	15:	IF bAutoModeOn AND bIUnitA_RowStopperEnd  THEN
		bQAUnitA_RowStopperMotorFwd2:=FALSE;
		CTU_2.RESET:=TRUE;
		 step:=step+1;
		END_IF

	16:	step:=step+1;

	17:	tRowStopperRevDly1(IN:=TRUE , PT:=t#1.5s , Q=> , ET=> );
		IF tRowStopperRevDly1.Q THEN bQAUnitA_RowStopperMotorFwd1:=FALSE; step:=step+1; END_IF

	18:	 step:=step+1;


	19:	IF bAutoModeOn   THEN
		bAConvSecStart:=TRUE;
		bQAUnitA_RowStopperMotorRev1:=TRUE;
		CTU_2.RESET:=FALSE;
		step:=step+1;
		END_IF

	20:	IF bAutoModeOn  AND bIUnitB_LiftPistonHome THEN
		CountResetBit1_24:=TRUE;
		step:=step+1;
		END_IF

	21:	IF bAutoModeOn  AND bIUnitA_RowStopperHome THEN
		bQAUnitA_RowStopperMotorRev1:=FALSE;
		sRetreivalAStatus:= 'IDLE';
		step:=step+1;
		END_IF

	22:	IF bAutoModeOn (* AND( UnitACompleteCheckCount.CV =  iATotalNoOfCones)*) THEN
		(*bUnitARowStopperStarted:=FALSE;
		UnitACompleteCheckCount.RESET:=TRUE;*);
		bQAUnitA_RowStopperMotorRev1:=FALSE;
		step:=0;
		END_IF

END_CASE


				              		(* ################### 2*4 Sequence for  Count Check ##################*)



CASE step2 OF

	0:	IF bUnitARowStopperStarted   AND bAutoModeOn  THEN
		F_TRIG_3_24(CLK:=bIUnitBConeCrossing , Q=> );
		IF F_TRIG_3_24.Q THEN TON_6(IN:= FALSE); step2:=step2+1; END_IF END_IF


	1:	TON_6(IN:= FALSE); TON_9(IN:= FALSE); step2:=step2+1;

	2:	 bAUnitBConeCrossing_1_24 :=TRUE;  step2:=Step2+1;

	3: 	TON_6(IN:=  TRUE  , PT:=t#100ms,Q=> , ET=> );
		IF TON_6.Q THEN bAUnitBConeCrossing_1_24:=FALSE;   step2:=step2+1; END_IF

	4:	IF   bIUnitBConeCrossing   THEN
		TON_9(IN:=  TRUE  , PT:=t#50ms,Q=> , ET=>);
		IF TON_9.Q THEN TON_6(IN:= FALSE);  step2:=step2+1; END_IF END_IF

	5:	TON_9(IN:= FALSE);
		step2:=0;

END_CASE


CASE step4 OF

	0:	IF bUnitARowStopperStarted    AND bAutoModeOn THEN
		F_TRIG_5(CLK:=bIUnitAConeCrossing , Q=> );
		IF F_TRIG_5.Q THEN TON_8(IN:= FALSE); step4:=step4+1; END_IF END_IF


	1:	TON_8(IN:= FALSE);
		TON_10(IN:= FALSE);
		step4:=step4+1;


	2:	 bAUnitAConeCrossing_1_24 :=TRUE;
		 step4:=step4+1;

	3: 	TON_8(IN:=  TRUE  , PT:=t#100ms,Q=> , ET=> );
		IF TON_8.Q   THEN  bAUnitAConeCrossing_1_24:=FALSE;  step4:=step4+1; END_IF

	4:	IF   bIUnitAConeCrossing   THEN
		TON_10(IN:=  TRUE  , PT:=t#50ms,Q=> , ET=>);
		IF TON_10.Q THEN TON_8(IN:= FALSE);  step4:=step4+1; END_IF END_IF

	5:	TON_8(IN:= FALSE);
		step4:=0;

END_CASE



UnitAConeCrossCount(
	CU:= bAUnitAConeCrossing_1_24   ,
	RESET:= ,
	PV:=3 ,
	Q=> ,
	CV=> );


UnitACompleteCheckCount(
	CU:=  bAUnitBConeCrossing_1_24   ,
	RESET:= ,
	PV:=iATotalNoOfCones ,
	Q=> ,
	CV=>UnitACompleteCheckCountCV );



						(*============= After 24 Cone Crossed the UnitB limit switch==============*)


IF UnitACompleteCheckCount.CV >=  iATotalNoOfCones AND CountResetBit1_24    THEN
 tConeCrossDly(IN:=TRUE , PT:=t#0.3s , Q=> , ET=> );  END_IF

IF tConeCrossDly.Q   THEN
tConeCrossDly_1_24(IN:=TRUE , PT:=t#1s , Q=> , ET=> );
UnitACompleteCheckCount.RESET:=TRUE;
bQAUnitA_RowStopperMotorFwd2:=FALSE;
bQAUnitA_RowStopperMotorFwd1:=FALSE;

IF tConeCrossDly_1_24.Q THEN
 bUnitARowStopperStarted:=FALSE;
UnitACompleteCheckCount.RESET:=TRUE;
 tConeCrossDly(IN:=FALSE);
tConeCrossDly_1_24(in:=FALSE);
CountResetBit1_24:=FALSE;
bQAUnitA_RowStopperMotorFwd2:=FALSE;
bQAUnitA_RowStopperMotorFwd1:=FALSE;
(*step:=0;*)
END_IF
IF tConeCrossDly_1_24.Q AND bIUnitA_RowStopperHome THEN
		bQAUnitA_RowStopperMotorRev1:=FALSE;
END_IF

END_IF


IF b2_3SetHmiSelected THEN iATotalNoOfCones:=18; END_IF
IF b2_4SetHmiSelected THEN iATotalNoOfCones:=24; END_IF

(*===============Stop Sequence===========*)


IF NOT bIEmergencySwitch OR bIMcStop OR bServoOff OR   bStopHmi THEN bStopRetUnitA:=TRUE;  UnitACompleteCheckCount.RESET:=TRUE;END_IF


IF bStopRetUnitA THEN
step:=0;
bAUnitAWeighOk:=FALSE;
bAConvFirstStart:=FALSE;
bQAUnitA_RowStopperMotorFwd1:=FALSE;
UnitAConeCrossCount.RESET:=FALSE;
bQAUnitA_RowStopperMotorFwd2:=FALSE;
bAConvSecStart:=FALSE;
bQAUnitA_RowStopperMotorRev1:=FALSE;
bRetUnitARst:=TRUE;
bUnitARowStopperStarted:=FALSE;
		UnitACompleteCheckCount.RESET:=FALSE;
step4:=0;
step2:=0;
END_IF

IF bIUnitA_RowStopperHome THEN
bStopRetUnitA:=FALSE;
bRetUnitARst:=FALSE;
END_IF

IF bRetUnitARst THEN
step4:=0;
step2:=0;
 END_IF


(***HMI Count***)

IF bUnitARowStopperStarted THEN
 RowStopperCountvalue:=UnitACompleteCheckCountCV;

ELSIF  NOT bUnitARowStopperStarted THEN
RowStopperCountvalue:=0;

END_IF
Count_Hmi:=RowStopperCountvalue;
END_PROGRAM

(* POU FunctionBlocks/SenSelect, ST *)
FUNCTION_BLOCK SenSelect
VAR_INPUT


	bVarIn1: BOOL;
	bVarIn2: BOOL;
	bVarIn3: BOOL;
	bVarIn4: BOOL;
END_VAR
VAR_OUTPUT


	ByteResult: USINT;
END_VAR
VAR

END_VAR
ByteResult.0:=bVarIn1;
ByteResult.1:=bVarIn2;
ByteResult.2:=bVarIn3;

ByteResult;
END_FUNCTION_BLOCK

(* POU Auto1/UnitB_RowStopper24, ST *)
PROGRAM UnitB_RowStopper24
VAR




	step: INT;
	bAUnitAWeighOk: BOOL;
	CTU_1: CTU;
	CTU_1Enable: BOOL;
	R_TRIG_1: R_TRIG;
	R_TRIG_2: F_TRIG;
	bQAUnitA_RowStopperMotorFwd1: BOOL;
	bQAUnitA_RowStopperMotorFwd2: BOOL;
	tRowStopperRevDly1: TON;
	bQAUnitA_RowStopperMotorRev1: BOOL;
	CTU_2: CTU;
	UnitBConeCount: CTU;
	CTU_1EnableUnitB: BOOL;
	temp1: BOOL;
	bStopRetUnitB: BOOL;
	bRetUnitBRst: BOOL;
	RowStopperMotorStopDly: TON;
	F_TRIG_3: F_TRIG;

	UnitBOverTemp: BOOL;
	bStartTemp1: BOOL;
	R_TRIG_5: R_TRIG;
	test: BOOL;
	bStopTemp2: BOOL;
	CTU_2CV: INT;
	CTU_test: CTU;
	R_TRIG_test: R_TRIG;
	InterLockStep: INT;

	CTU_2Enable: BOOL;
	timer1: TON;
	UnitBCompleteCheckCountCV: INT;
	Ctu_2_Rst: BOOL;
	F_TRIG_1: F_TRIG;
	bRestBit: BOOL;
	bResetBit: BOOL;
	R_TRIG_6: R_TRIG;
	timer2: TON;
	SenSelect_2: SenSelect;
	iSensorOnVal: UINT;
	iAConeCrossCount1: INT;
	GetDLy: TON;
	bCheckSensor1: BOOL;
	step2: INT;
	TON_9: TON;
	TON_6: TON;
	tConeCrossDly: TON;
	bAUnitBConeCrossing_24_B: BOOL;
	tConeCrossDly_2_24: TON;
	CountResetBit2_24: BOOL;
END_VAR
(*=============Checking the No of sensors sensed================*)

IF bCheckSensor1 THEN
SenSelect_2(
		bVarIn1:=bIUnitBConedetection1 ,
		bVarIn2:= bIUnitBConedetection2,
		bVarIn3:= bIUnitBConedetection3,
		ByteResult=>iSensorOnVal );
END_IF

IF iSensorOnVal=7 THEN iAConeCrossCount1:=3;
	ELSIF  iSensorOnVal=6 THEN iAConeCrossCount1:=2;
	ELSIF  iSensorOnVal=5 THEN iAConeCrossCount1:=2;
	ELSIF  iSensorOnVal=4 THEN iAConeCrossCount1:=1;
	ELSIF  iSensorOnVal=3 THEN iAConeCrossCount1:=2;
	ELSIF  iSensorOnVal=2 THEN iAConeCrossCount1:=1;
	ELSIF  iSensorOnVal=1 THEN iAConeCrossCount1:=1;
END_IF


bQAUnitB_RowStopperMotorForward:=( bQAUnitB_RowStopperMotorFwd1 OR bQAUnitB_RowStopperMotorFwd2  );

bQAUnitB_RowStopperMotorReverse:= ( bQAUnitB_RowStopperMotorRev1 OR bRetUnitBRst  );


CASE step OF

	0:	IF bAutoModeOn AND bAUnitBWeighOk  AND bRetUnitBStart  AND NOT bStopEnable AND bAinterlockinit   THEN
		UnitBConeCrossCount.RESET:=TRUE;
		CTU_2.RESET:=TRUE;
		UnitBCompleteCheckCount_24.RESET:=TRUE;
		CountResetBit2_24 :=FALSE;
		step:=step+1;
		END_IF

	1:	 step:=step+1;

	2:	IF bAutoModeOn   AND  UnitBCompleteCheckCount_24.CV = 0 AND NOT CountResetBit2_24 THEN
		CTU_2.RESET:=FALSE;
		UnitBConeCrossCount.RESET:=FALSE;
		UnitBCompleteCheckCount_24.RESET:=FALSE;
		step:=step+1;
		END_IF


	3:	bRestBit:=TRUE;
		step:=step+1;


	4:	IF bAutoModeOn  AND NOT bIUnitBConedetection1 AND NOT bIUnitBConedetection2 AND NOT bIUnitBConedetection3
		AND NOT bUnitARowStopperStarted AND NOT bAMainIntStarted  AND NOT bStopEnable AND NOT bAPauseSeq THEN
		timer1(IN:=FALSE);
		timer2(IN:=FALSE);
		bAConvFirstStartUnitB:=TRUE;
		bQAUnitB_RowStopperMotorFwd1:=TRUE;
		bAUnitBWeighOk:=FALSE;
		bRetUnitBStart:=FALSE;
		sRetreivalBStatus:= 'Running';
		bUnitBRowStopperStarted:=TRUE;
		step:=step+1;
		ELSIF   bIUnitB_RowStopperEnd  THEN  step:=12;
		END_IF

	5:	RowStopperMotorStopDly(In:=FALSE); step:=step+1;


	6:	IF bIUnitBConedetection1 OR  bIUnitBConedetection2  OR  bIUnitBConedetection3 THEN
		UnitBConeCount.RESET:=TRUE;
		step:=step+1;
		ELSIF NOT bIUnitBConedetection1 AND NOT  bIUnitBConedetection2 AND NOT  bIUnitBConedetection3 AND bIUnitB_RowStopperEnd THEN
		step:=15;
		END_IF

	7:	RowStopperMotorStopDly( IN:=TRUE , PT:=T#0.5S , Q=> , ET=> );IF RowStopperMotorStopDly.Q   THEN  step:=step+1; END_IF


	8:	UnitBConeCount.RESET:=FALSE;
		bQAUnitB_RowStopperMotorFwd1:=FALSE;
		tRowStopperRevDly1(IN:=FALSE);
		step:=step+1;

	9:	IF NOT bAPauseSeq THEN bCheckSensor1:=TRUE;  step:=step+1; END_IF

	10:	GetDLy(IN:=TRUE , PT:=t#0.6s , Q=> , ET=> );
		 IF GetDLy.Q THEN bCheckSensor1:=FALSE;   step:=step+1;
		END_IF


	11:	IF  (UnitBConeCount.CV=iAConeCrossCount1)  AND NOT bIUnitB_RowStopperEnd THEN
		RowStopperMotorStopDly(In:=FALSE);
		 step:=4;
		ELSE
		IF bIUnitB_RowStopperEnd THEN
		    step:=step+1;
		END_IF END_IF



	12:	IF NOT bAPauseSeq THEN tRowStopperRevDly1(IN:=FALSE); step:=step+1; END_IF

	13:	IF bAutoModeOn    (* AND NOT bQAFeedingConveyorMotor *) THEN
		bQAUnitB_RowStopperMotorFwd2:=TRUE;
		step:=step+1;
		END_IF


	14:	 step:=step+1;

	15:	IF bAutoModeOn AND bIUnitB_RowStopperEnd THEN
		bQAUnitB_RowStopperMotorFwd2:=FALSE;
		bQAUnitB_RowStopperMotorFwd1:=FALSE;
		UnitBConeCount.RESET:=TRUE;
		CTU_2.RESET:=TRUE;
		 step:=step+1;
		END_IF

	16:	  step:=step+1;

	17:	tRowStopperRevDly1(IN:=TRUE , PT:=t#1.5s , Q=> , ET=> );
		IF tRowStopperRevDly1.Q THEN step:=step+1; END_IF

	18:	step:=step+1;

	19:	IF bAutoModeOn  THEN
		bAConvSecStartUnitB:=TRUE;
		CTU_2.RESET:=FALSE;
		UnitBConeCount.RESET:=FALSE;
		bQAUnitB_RowStopperMotorRev1:=TRUE;
		step:=step+1;
		END_IF

	20:	IF bAutoModeOn  AND bIUnitB_LiftPistonEnd THEN
		CountResetBit2_24:=TRUE;
		step:=step+1;
		END_IF


	21:	IF bAutoModeOn  AND bIUnitB_RowStopperHome THEN
		bQAUnitB_RowStopperMotorRev1:=FALSE;
		sRetreivalBStatus:= 'IDLE';
		step:=step+1;
		END_IF

	22:	IF bAutoModeOn  (*AND (UnitBCompleteCheckCount_24.CV >=  iATotalNoOfCones)*) THEN
 		(*bUnitBRowStopperStarted:=FALSE;
		UnitBCompleteCheckCount_24.RESET:=FALSE;*)
		step:=0;
		END_IF



END_CASE


					(* ######################### 2*4 Cone Count Sequence ####################*)




CASE step2 OF

	0:	IF bUnitBRowStopperStarted  AND bAutoModeOn THEN
		F_TRIG_3(CLK:=bIUnitBConeCrossing , Q=> );
		IF F_TRIG_3.Q THEN TON_6(IN:= FALSE); step2:=step2+1; END_IF END_IF


	1:	TON_6(IN:= FALSE);
		TON_9(IN:= FALSE);
		step2:=step2+1;


	2:	 bAUnitBConeCrossing_24_B :=TRUE;
		 step2:=Step2+1;

	3:	 step2:=step2+1;

	4: 	TON_6(IN:=  TRUE  , PT:=t#100ms,Q=> , ET=> );
		IF TON_6.Q THEN bAUnitBConeCrossing_24_B:=FALSE;   step2:=step2+1; END_IF


	5:	 step2:=step2+1;

	6:	IF   bIUnitBConeCrossing THEN
		TON_9(IN:=  TRUE  , PT:=t#50ms,Q=> , ET=>);
		IF TON_9.Q THEN TON_6(IN:= FALSE);  step2:=step2+1; END_IF END_IF


	7:	 step2:=step2+1;

	8:	 step2:=step2+1;

	9:	 step2:=step2+1;

	10:	TON_9(IN:= FALSE);
		step2:=0;


END_CASE




UnitBConeCount(
	CU:= ( bAUnitBConeCrossing_24_B)  ,
	RESET:= ,
	PV:=3 ,
	Q=> ,
	CV=> );

UnitBCompleteCheckCount_24(
	CU:= bAUnitBConeCrossing_24_B  ,
	RESET:= ,
	PV:=iATotalNoOfCones ,
	Q=> ,
	CV=>UnitBCompleteCheckCountCV );

(*============= After 18 Cone Crossed the UnitB limit switch==============*)

IF UnitBCompleteCheckCount_24.CV >=  iATotalNoOfCones AND CountResetBit2_24  AND bAutoModeOn  THEN
 tConeCrossDly(IN:=TRUE , PT:=t#0.3s , Q=> , ET=> );
END_IF

IF tConeCrossDly.Q THEN
tConeCrossDly_2_24(IN:=TRUE , PT:=t#1s , Q=> , ET=> );
UnitBCompleteCheckCount_24.RESET:=TRUE;

IF tConeCrossDly_2_24.Q THEN
 bUnitBRowStopperStarted:=FALSE;
UnitBCompleteCheckCount_24.RESET:=TRUE;
  tConeCrossDly(IN:=FALSE);
tConeCrossDly_2_24(in:=FALSE);
CountResetBit2_24:=FALSE;
 END_IF
ELSE
UnitBCompleteCheckCount.RESET:=FALSE;

END_IF







(*===============Stop Sequence===========*)


IF NOT bIEmergencySwitch OR bIMcStop OR bServoOff OR  bStopHmi THEN bStopRetUnitB:=TRUE; END_IF


IF bStopRetUnitB THEN
step:=0;
bAUnitBWeighOk:=FALSE;
bAConvFirstStartUnitB:=FALSE;
bQAUnitB_RowStopperMotorFwd1:=FALSE;
UnitBConeCount.RESET:=FALSE;
bQAUnitB_RowStopperMotorFwd2:=FALSE;
bAConvSecStartUnitB:=FALSE;
bQAUnitB_RowStopperMotorRev1:=FALSE;
bRetUnitBRst:=TRUE;
bUnitBRowStopperStarted:=FALSE;
step2:=0;
END_IF

IF bIUnitB_RowStopperHome THEN
bStopRetUnitB:=FALSE;
bRetUnitBRst:=FALSE;
END_IF



IF bAutoModeOn  AND  bResetBit AND bIUnitBConedetection1 AND bIUnitBConedetection3 AND bIUnitBConedetection3
AND NOT  bIUnitB_RowStopperHome THEN Ctu_2_Rst:=TRUE;  ELSE Ctu_2_Rst:= FALSE; END_IF

R_TRIG_6(CLK:=Ctu_2_Rst , Q=> );

CTU_2.RESET:= R_TRIG_6.Q;


(***HMI Count***)

IF bUnitBRowStopperStarted THEN
CountB_Hmi:=UnitBCompleteCheckCountCV;
ELSIF  NOT bUnitBRowStopperStarted THEN
CountB_Hmi:=0;
END_IF
END_PROGRAM

(* POU Auto/OneMinConv, ST *)
	PROGRAM OneMinConv
VAR
	bQAGrossWtPiston1: BOOL;
	bQARollerConvMotor1: BOOL;
	step: INT;
	Timer1: TON;
	Timer2: TON;

	Timer3: TON;
	bQARollerConvMotor2: BOOL;
	bAPartCount: BOOL;
	R_TRIG_1: R_TRIG;
	PartCounter: CTU;
	rGrossWtTolMax: REAL;
	rGrossWtTolMin: REAL;
	bGrossWieghtOkTemp: BOOL;
	rGrossWeighToReportTemp: STRING;
	iTotalpartCounttemp: DINT;
END_VAR
	bQAGrossWtPiston:= bQAGrossWtPiston1 ;
	bQARollerConvMotor:=bQARollerConvMotor1 OR bQARollerConvMotor2 ;


rGrossWtTolMax:= (sSettingArray[i].iGrosswt + sSettingArray[i].iGrossTol);

rGrossWtTolMin:= (sSettingArray[i].iGrosswt - sSettingArray[i].iGrossTol);


CASE step OF

	0:	IF bAutoModeOn AND bAOneMinConvStart   AND NOT bAPauseSeq THEN
		bQARollerConvMotor1:=TRUE;
		Timer1(IN:=FALSE);
		Timer2(IN:=FALSE);
		Timer3(IN:=FALSE);
		 step:=step+1;
		END_IF

	1:	IF bIGrossWtDeductSensor THEN
		bQARollerConvMotor1:=FALSE;
		bAOneMinConvStart:=FALSE;
		 step:=step+1;
		END_IF

	2:	Timer1(IN:=TRUE , PT:=t#1s , Q=> , ET=> );
		IF Timer1.Q THEN step:= step+1; END_IF   (*====== Modified for  Gross  Weight   bypass  then removed  ==============*)

	3:	bQAGrossWtPiston1:=TRUE;
		IF bIGrossWtPistonEnd  AND NOT bAGrossWtSenRsError THEN step:=step+1; END_IF

	4:	 tGrossWtCheckDly(IN:=FALSE);
		Timer2(IN:=TRUE , PT:=t#1s , Q=> , ET=> );
		IF Timer2.Q THEN step:=step+1; END_IF

	5:	bReadGWieght:=TRUE;
		step:=step+1;


	6:	IF bReadGWieght THEN
		tGrossWtCheckDly(IN:=TRUE , PT:=t#9.5s , Q=> , ET=> );
		IF tGrossWtCheckDly.Q THEN 	step:=step+1;END_IF
		END_IF


	7:	IF  rGrossWeight >=rGrossWtTolMin  AND   rGrossWeight  <= rGrossWtTolMax  THEN
		bGrossWieghtOkTemp:=TRUE; rGrossWeighToReport:=rGrossWeight ;  bGrossWieghtNokTemp:=FALSE;
		step:=step+1;
		ELSIF  rGrossWeight  >= rGrossWtTolMax THEN
		bGrossWieghtNokTemp:=TRUE; bGrossWieghtOkTemp:=FALSE;
		step:=step+2;
		ELSIF   rGrossWeight  <=rGrossWtTolMin   THEN
		bGrossWieghtNokTemp:=TRUE; bGrossWieghtOkTemp:=FALSE;
		step:=step+2;
		END_IF


	8:	IF bGrossWieghtOkTemp THEN bGrossWieghtOk:=TRUE; bQAGrossWieghtOkIndi:=TRUE; step:=step+2;  END_IF

	9:	IF bGrossWieghtNokTemp THEN bGrossWieghtNOk:=TRUE; bReadGWieght:=FALSE; step:=step+2; END_IF


	10:	IF bGrossWieghtOk (*  AND NOT bGrossWieghtNok *) AND bAutoModeOn  AND NOT bAPauseSeq THEN bQAGrossWtPiston1:=FALSE; bReadGWieght:=FALSE; bGrossWieghtOkTemp:=FALSE; bQAGrossWieghtOkIndi:=FALSE;   (*====== Modified for  Gross  Weight   bypass  ==============*)
		bACyclePass:=TRUE;
		GrossWtReedSwBit:=TRUE;
		step:=step+2;
		 END_IF

	11:	IF bErrorReset THEN  bGrossWieghtNOk:=FALSE;  step:=4; END_IF

	12:	IF bIGrossWtPistonHome  AND NOT bAGrossWtHomeSenRsError THEN GrossWtReedSwBit:=FALSE ;step:=step+1;END_IF

	13:	bACyclePass:=FALSE;
		 step:=step+1;

	14:	IF NOT   bAPauseSeq  THEN
		bQARollerConvMotor2:=TRUE;
		bReadGWieght:=FALSE;
		Step:=Step+1;
	(*	Timer3(IN:=TRUE , PT:=t#30s , Q=> , ET=> );
		IF Timer3.Q THEN step:=step+1; END_IF    *)
		END_IF


	15:	IF NOT  bIGrossWtDeductSensor THEN
		bQARollerConvMotor2:=FALSE;
		 bOneMinConvOver:=TRUE;

		step:=0;
		END_IF

END_CASE

sFinalGrossWt:=MID(STR:=rGrossWeighToReportTemp, LEN:=7, POS:=1);

rGrossWeighToReportTemp:=REAL_TO_STRING (rGrossWeight);

IF bGrossWieghtOk THEN var_7:= sFinalGrossWt ; END_IF

(*=====Carton Completed Count Logic=========*)

	IF bACyclePass AND bAutoModeOn THEN bAPartCount:=TRUE; ELSE bAPartCount:=FALSE; END_IF


R_TRIG_1(CLK:=bAPartCount , Q=> );
PartCounter(
	CU:=R_TRIG_1.Q ,
	RESET:=bSaveRecipeHmi ,
	PV:= 9999,
	Q=> ,
	CV=> );

iTotalpartCountTemp:=PartCounter.CV;

ITotalSample:=iTotalpartCountTemp;
(*========== No Of Cartons Processed Logic==========*)

IF b2_3SetHmiSelected AND bACyclePass THEN   iTotalCones := ( iTotalpartCountTemp  * 18 );  iTotalpartCount:=iTotalpartCountTemp;

ELSIF b2_4SetHmiSelected  AND bACyclePass THEN  iTotalCones := ( iTotalpartCountTemp  * 24  );  iTotalpartCount:=iTotalpartCountTemp;

END_IF


IF NOT bIEmergencySwitch OR   bStopHmi   OR bServoOff  OR bIMcStop  THEN
step:=0;
bReadGWieght:=FALSE;
bAOneMinConvStart:=FALSE;
bQARollerConvMotor1:=FALSE;
bQARollerConvMotor2:=FALSE;
bQAGrossWtPiston1:=FALSE;
bGrossWieghtNOk:=FALSE;
bACyclePass:=FALSE;
Timer1(IN:=FALSE);
Timer2(IN:=FALSE);
Timer3(IN:=FALSE);
tGrossWtCheckDly(IN:=FALSE);
END_IF
END_PROGRAM

(* POU Auto/Sealing_Unit, ST *)
PROGRAM Sealing_Unit
VAR
	step: INT;
	tA3ConeStartDly: TON;
	tA3ConeSealCompDly: TON;
	test: BOOL;

END_VAR
IF NOT bIEmergencySwitch OR  bStopHmi    OR bServoOff OR bIMcStop   THEN
	tA3ConeStartDly(IN:=FALSE);
	tA3ConeSealCompDly(IN:=FALSE);
	bQASealingSeparatorYAxisPistonValve:=FALSE;
	bQASealingTopPistonValve:=FALSE;
	bQASealingSeparatorXAxisPistonValve:=FALSE;
	bA3ConeWrappOver:=FALSE;
	bA3ConeWrappOver_24:=FALSE;
	bA4thWrappOver:=FALSE;
	bA6thConeWrappOver:=FALSE;
	bA8thConeWrappOver:=FALSE;
	bA6ConeWrappOver23:=FALSE;
	bMManualSealOn:=FALSE;
	bQMSealingTopPistonValve:=FALSE;
	Step:=0;
	SealingOver1:=FALSE;
	bA3ConeWrappOver_24:=FALSE;
END_IF


CASE step OF

	0:	IF b2_4SetHmiSelected OR b2_3SetHmiSelected  AND bAutoModeOn  THEN
		Step:=step+1;
		END_IF

	1:	step:=step+1;


	2:	IF bAutoModeOn AND  bA3ConeWrappOver  OR bA4thWrappOver OR bA6thConeWrappOver  OR bA8thConeWrappOver  OR bA6ConeWrappOver23
		OR bA3ConeWrappOver_24 AND NOT bAPauseSeq THEN
		tA3ConeStartDly(IN:=TRUE , PT:=t#1s , Q=> , ET=> );
		IF tA3ConeStartDly.Q THEN  step:=step+1; END_IF
		END_IF

	3:	IF bIWrappingChannelPiston1_Home AND bIWrappingChannelPiston2_Home  AND bIWrappingChannelPiston3_Home THEN
		step:=step+1;END_IF    sMessage_Sealing:='Check Wrapping Piston Home 1 & 2 & 3 Reed Switch';


	4:	IF bAutoModeOn AND   bISealingBottomPistonHome  AND bISealingTopPistonHome AND bISealingSeparatorXAxisHome
		AND bISealingSeparatorYAxisHome   AND  NOT bAPauseSeq THEN
		bQASealingSeparatorYAxisPistonValve:=TRUE;
		tA3ConeSealCompDly(IN:=FALSE);
		 step:=step+1;
		END_IF  sMessage_Sealing:='Check All  Piston Home  Reed Switch';

	5:	 step:=step+1;

	6:	IF bAutoModeOn AND  bISealingSeparatorYAxisEnd AND  NOT bAPauseSeq  AND NOT bASealSepaY_axisRsError  THEN
		tA3ConeStartDly(IN:=FALSE);
		bQASealingTopPistonValve:=TRUE;
		step:=step+1;
		END_IF

	7:	step:=step+1;

	8:	IF bAutoModeOn AND  bISealingTopPistonEnd AND bISealingBottomPistonEnd  THEN
		tA3ConeSealCompDly(IN:=TRUE, PT:= SealComDlyTemp, Q=> , ET=> );
		IF tA3ConeSealCompDly.Q THEN   step:=step+1; END_IF
		END_IF

	9:	step:=step+1;

	10:	IF bAutoModeOn AND  bISealingTopPistonEnd AND bISealingBottomPistonEnd AND bISealingSeparatorYAxisEnd AND  NOT bAPauseSeq
		  AND NOT SealTopBottomRsError THEN
		bQASealingSeparatorXAxisPistonValve:=TRUE;
		step:=step+1;
		END_IF  sMessage_Sealing:='Check Sealing Top, Bottom, Separator YAxis  Piston End  Reed Switch';

	11:	 step:=step+1;

	12:	IF bAutoModeOn AND  bISealingSeparatorXAxisEnd AND  NOT bAPauseSeq  AND  NOT bASealSepaX_axisRsError THEN
		step:=step+1;
		 END_IF

	13:	 step:=step+1;

	14:	bQASealingTopPistonValve:=FALSE;
		bA3ConeWrappOver:=FALSE;
		bA3ConeWrappOver_24:=FALSE;
		bA4thWrappOver:=FALSE;
		bA6thConeWrappOver:=FALSE;
		bA8thConeWrappOver:=FALSE;
		bA6ConeWrappOver23:=FALSE;
		bQASealingSeparatorYAxisPistonValve:=FALSE;
		bQASealingSeparatorXAxisPistonValve:=FALSE;
		step:=step+1;

	15:	step:=step+1;

	16:	IF b2_4SetHmiSelected THEN step:=step+1; ELSIF b2_3SetHmiSelected THEN step:=step+1; END_IF


	17:	IF bAutoModeOn AND NOT bA3ConeWrappOver AND NOT bA4thWrappOver AND NOT bA6thConeWrappOver AND NOT bA8thConeWrappOver
		AND NOT bA3ConeWrappOver_24 AND bISealingSeparatorXAxisHome AND  bISealingTopPistonHome AND bISealingBottomPistonHome
		AND bISealingSeparatorYAxisHome  THEN
		SealingOver1:=TRUE; step:=step+1;
		END_IF sMessage_Sealing:='Check All Piston Home  Reed Switch';


	18:	IF bAutoModeOn AND bISealingSeparatorXAxisHome AND  bISealingTopPistonHome AND bISealingBottomPistonHome AND bISealingSeparatorYAxisHome
		THEN
		 step:=step+1;
		END_IF sMessage_Sealing:='Check All Piston Home  Reed Switch';

	19:	step:=step+1;

	20:	 step:=step+1;

	21:	step:=0;



END_CASE



IF bAutoModeOn AND NOT bA3ConeWrappOver AND NOT bA4thWrappOver AND NOT bA6thConeWrappOver AND NOT bA8thConeWrappOver AND
 bISealingSeparatorXAxisHome AND  bISealingTopPistonHome AND bISealingBottomPistonHome AND bISealingSeparatorYAxisHome  THEN
SealingSafety:=TRUE; ELSE SealingSafety:=FALSE;END_IF
END_PROGRAM

(* POU New Folder/ConeAllignAlarm, ST *)
PROGRAM ConeAllignAlarm
VAR
	ConeMiss: INT;
	TON_1: TON;
	TON_2: TON;
	TON_3: TON;
	Timer_4: TON;

	bAConeMissErrorAtWrpConvTemp: BOOL;
	bNotSensing: BOOL;
	bNotSensingtEMP: BOOL;

	TON_3_24: TON;
	TON_12: TON;

END_VAR
(*...................Cone Allignment Alarm.....................*)


IF bQAWrappingConveyorMotor1 AND b2_3SetHmiSelected THEN TON_3(IN:=TRUE , PT:= t#7s, Q=> , ET=> );  ELSE  TON_3(IN:=FALSE); END_IF

IF  bAutoModeOn AND TON_3.Q AND NOT bIWrappingCone1 AND b2_3SetHmiSelected  THEN
 bAConeMissErrorAtWrpConvTemp:=TRUE;  END_IF

IF bAutoModeOn  AND bIWrappingCone1 AND b2_3SetHmiSelected THEN
bAConeMissErrorAtWrpConvTemp:=FALSE; END_IF     (*Change*)

IF bErrorReset AND b2_3SetHmiSelected THEN
TON_3(IN:=FALSE); bAConeMissErrorAtWrpConvTemp:=FALSE;  END_IF

IF NOT bIEmergencySwitch OR bStopHmi  OR bServoOff OR bIMcStop  AND b2_3SetHmiSelected  THEN
bAConeMissErrorAtWrpConvTemp:=FALSE;
ConeMissAlarm:='';
 TON_3(IN:=FALSE);
END_IF


(* ================== Cone Missing 2 & 3 Logic on Wrapping Conveyor===============*)

IF bWrapConvStopped2 AND b2_3SetHmiSelected  AND  NOT bAPauseSeq  THEN Timer_4(IN:=TRUE , PT:=t#4s , Q=> , ET=> ); ELSE  Timer_4(IN:=FALSE); END_IF

IF bAutoModeOn  AND  Timer_4.Q AND  (NOT bIWrappingCone1 OR NOT bIWrappingCone2 OR NOT bIWrappingCone3 ) AND NOT bConeMiss2AtWrapConvtEMP
AND b2_3SetHmiSelected  THEN bConeMiss2AtWrapConvtEMP:=TRUE;
ELSE
 IF  bAutoModeOn AND b2_3SetHmiSelected AND bWrapConvStopped2   AND bIWrappingCone1 AND bIWrappingCone2 AND bIWrappingCone3 THEN
  TON_12(IN:=TRUE , PT:= t#0.7s, Q=> , ET=> );  Timer_4(IN:=FALSE);

IF TON_12.Q AND b2_3SetHmiSelected THEN  bWrapConvStopped2:=FALSE; END_IF
 END_IF  END_IF


IF bErrorReset  AND bConeMiss2AtWrapConvtEMP AND  bIWrappingCone1 AND bIWrappingCone2 AND bIWrappingCone3
 THEN Timer_4(IN:=FALSE); TON_12(in:=FALSE); bConeMiss2AtWrapConvtEMP:=FALSE;
bAByPassOn:=TRUE;  bConeMiss2AtWrapConv:=FALSE; bConeMiss2AtWrapConvtEMP:=FALSE; ConeMissAlarm:=''; END_IF


IF NOT bIEmergencySwitch OR bIMcStop OR bStopHmi OR bServoOff THEN
bWrapConvStopped2:=FALSE;
bConeMiss2AtWrapConvtEMP:=FALSE;
bCount_ConvLockBit:=FALSE;
Timer_4(IN:=FALSE);
END_IF



(*============Wrapping Cone Missing Msg to Hmi=============*)

IF bAConeMissErrorAtWrpConvTemp AND b2_3SetHmiSelected THEN
ConeMissAlarm:='Allign the Cone  on Wrapping Conveyer ';
ELSIF bConeMiss2AtWrapConvtEMP AND b2_3SetHmiSelected  THEN
ConeMissAlarm:='Allign the Cone  on Wrapping Conveyer ';
ELSIF bConeMiss3AtWrapConv  AND b2_3SetHmiSelected THEN
ConeMissAlarm:='Allign the Cone  on Wrapping Conveyer ';
ELSIF bConeMiss4AtWrapConv AND b2_3SetHmiSelected  THEN
ConeMissAlarm:='Allign the Cone  on Wrapping Conveyer ';

ELSIF bACheckWrappConvError1_23 AND b2_3SetHmiSelected  THEN
ConeMissAlarm:='Check Wrapping Sensor 1 & 2 & 3';
ELSIF bACheckWrappConvError2  AND b2_3SetHmiSelected THEN
ConeMissAlarm:='Check Wrapping Sensor  2 & 3';
ELSIF bACheckWrappConvError3 AND b2_3SetHmiSelected THEN
ConeMissAlarm:='Check Wrapping Sensor 1 & 2 & 3';
ELSIF bACheckWrappConvError4 AND b2_3SetHmiSelected THEN
ConeMissAlarm:='Check Wrapping Sensor  3';
ELSIF NOT bConeMiss1AtWrapConv  AND NOT bAConeMissErrorAtWrpConvTemp AND NOT  bConeMiss2AtWrapConvtEMP AND NOT bConeMiss3AtWrapConv
AND NOT bConeMiss4AtWrapConv AND NOT  bACheckWrappConvError1_23 AND NOT bACheckWrappConvError2 AND NOT bACheckWrappConvError3
 AND NOT bACheckWrappConvError4 THEN
ConeMissAlarm:='   ';
END_IF


IF( bAConeMissErrorAtWrpConvTemp OR bConeMiss1AtWrapConv OR bConeMiss2AtWrapConvtEMP OR bConeMiss3AtWrapConv OR  bConeMiss4AtWrapConv)
 AND b2_3SetHmiSelected  THEN  bAConeMissErrorAtWrpConv:=TRUE; ELSE bAConeMissErrorAtWrpConv:=FALSE; END_IF


IF (bConeMiss1AtWrapConv OR bConeMiss2AtWrapConv OR bConeMiss3AtWrapConv OR  bConeMiss4AtWrapConv  OR bAConeMissErrorAtWrpConv
 OR bAConeMissErrorAtWrpConv OR bACheckWrappConvError1_23 OR bACheckWrappConvError4 OR bACheckWrappConvError2 OR bACheckWrappConvError3)
 AND b2_3SetHmiSelected
THEN bHmiColourChangeBit2:=TRUE; ELSE  bHmiColourChangeBit2:=FALSE; END_IF




(* ================== Cone Missing 4 & 5 Logic on Wrapping Conveyor===============*)

IF bWrapConvStopped3 AND b2_3SetHmiSelected  THEN Timer_5(IN:=TRUE , PT:=t#4s , Q=> , ET=> ); ELSE  Timer_5(IN:=FALSE); END_IF

IF bAutoModeOn  AND  Timer_5.Q AND  (NOT bIWrappingCone1 OR NOT bIWrappingCone2 (*OR NOT bIWrappingCone3 *)) AND NOT bConeMiss3AtWrapConv
AND b2_3SetHmiSelected  THEN bConeMiss3AtWrapConv:=TRUE;
ELSE
 IF  bAutoModeOn AND b2_3SetHmiSelected AND bWrapConvStopped3   AND bIWrappingCone1 AND bIWrappingCone2 (*AND bIWrappingCone3*) THEN
  TON_12_2_3(IN:=TRUE , PT:= t#3s, Q=> , ET=> );  (*Timer_5(IN:=FALSE);*)

IF TON_12_2_3.Q AND b2_3SetHmiSelected THEN  bWrapConvStopped3:=FALSE; END_IF
 END_IF  END_IF


(*
IF bAutoModeOn AND bWrapConvStopped3 AND bIWrappingCone1  AND b2_3SetHmiSelected  AND NOT bConeMiss3AtWrapConv
THEN  bWrapConvStopped3:=FALSE;   (*========need to give push cyl output=========*)

ELSIF bAutoModeOn AND b2_3SetHmiSelected  AND Timer_5.Q  AND NOT  bIWrappingCone1  THEN bConeMiss3AtWrapConv:=TRUE;

END_IF
*)

 IF bConeMiss3AtWrapConv AND bAutoModeOn  AND b2_3SetHmiSelected AND bIWrappingCone1 AND   bIWrappingCone2 AND bErrorReset
AND NOT bIWrappingCone3 THEN
 bAByPassOn2:=TRUE;  bConeMiss3AtWrapConv:=FALSE;Timer_5(IN:=FALSE); TON_12_2_3(IN:=FALSE);
 END_IF

IF NOT bIEmergencySwitch OR bIMcStop OR bStopHmi OR  bServoOff THEN
bWrapConvStopped3:=FALSE;
bConeMiss3AtWrapConv:=FALSE;
Timer_5(IN:=FALSE);
TON_12_2_3(IN:=FALSE);
END_IF

(* ==================   6th Cone Missing Logic on Wrapping Conveyor===============*)

IF bWrapConvStopped4 AND b2_3SetHmiSelected  THEN Timer_6(IN:=TRUE , PT:=t#4s , Q=> , ET=> ); ELSE  Timer_6(IN:=FALSE); END_IF

IF bAutoModeOn  AND  Timer_6.Q AND  (NOT bIWrappingCone1 OR NOT bIWrappingCone2 OR NOT bIWrappingCone3 ) AND NOT bConeMiss4AtWrapConv
AND b2_3SetHmiSelected  THEN bConeMiss4AtWrapConv:=TRUE;
ELSE
 IF  bAutoModeOn AND b2_3SetHmiSelected AND bWrapConvStopped4   AND bIWrappingCone1 AND bIWrappingCone2 AND bIWrappingCone3 THEN
  TON_13_2_3(IN:=TRUE , PT:= t#1s, Q=> , ET=> );  Timer_6(IN:=FALSE);

IF TON_13_2_3.Q AND b2_3SetHmiSelected THEN  bWrapConvStopped4:=FALSE; END_IF
 END_IF  END_IF

(*

IF bAutoModeOn  AND b2_3SetHmiSelected AND bWrapConvStopped4 AND bIWrappingCone1 AND bIWrappingCone2 AND bIWrappingCone3   AND NOT bConeMiss4AtWrapConv
THEN bAWrapConeCyl123_23:=TRUE;  bWrapConvStopped4:=FALSE;   (*========need to give push cyl output=========*)

ELSIF bAutoModeOn  AND b2_3SetHmiSelected AND Timer_6.Q  AND( NOT  bIWrappingCone1 OR NOT bIWrappingCone2 OR NOT bIWrappingCone3 )
 THEN bConeMiss4AtWrapConv:=TRUE; bCount_ConvLockBitTemp:=TRUE;

END_IF*)

(* ==================Error Acknlodge for  Cone Missing Logic on Wrapping Conveyor===============*)


 IF bConeMiss4AtWrapConv  AND b2_3SetHmiSelected AND bAutoModeOn AND bIWrappingCone1 AND   bIWrappingCone2 AND  bIWrappingCone3  AND bErrorReset
THEN bAByPassOn3:=TRUE;  bConeMiss4AtWrapConv:=FALSE; Timer_6(IN:=FALSE); TON_13_2_3(IN:=FALSE);END_IF


IF NOT bIEmergencySwitch OR bIMcStop OR bStopHmi OR  bServoOff THEN
bWrapConvStopped4:=FALSE;
Timer_6(IN:=FALSE);
TON_13_2_3(IN:=FALSE);
bConeMiss4AtWrapConv:=FALSE;
bCount_ConvLockBitTemp:=FALSE;
bAByPassOn2:=FALSE;
END_IF


								(*######################      2*4  Alarm ####################*)


IF b2_4SetHmiSelected THEN

IF (bACheckWrappConvError1 OR bACheckWrappConvError2 OR bACheckWrappConvError3 OR  bACheckWrappConvError4  OR bACheckWrappConvError5 OR
 bAConeMissErrorAtWrpConvTemp1_24 OR bAConeMissErrorAtWrpConvTemp2_24 OR bAConeMissErrorAtWrpConvTemp3_24 OR bAConeMissErrorAtWrpConvTemp4_24
 OR  bAConeMissErrorAtWrpConvTemp5_24   ) AND b2_4SetHmiSelected  THEN
		 bHmiColourChangeBit2:=TRUE;
ELSE	 bHmiColourChangeBit2:=FALSE; END_IF

IF (bAConeMissErrorAtWrpConvTemp1_24 OR bAConeMissErrorAtWrpConvTemp2_24 OR bAConeMissErrorAtWrpConvTemp3_24 OR bAConeMissErrorAtWrpConvTemp4_24
 OR  bAConeMissErrorAtWrpConvTemp5_24 ) AND b2_4SetHmiSelected THEN
		 bAConeMissErrorAtWrpConv:=TRUE;
 ELSE 	 bAConeMissErrorAtWrpConv:=FALSE; END_IF

IF bACheckWrappConvError1 OR  bACheckWrappConvError2 OR  bACheckWrappConvError3 OR  bACheckWrappConvError4 OR  bACheckWrappConvError5 THEN
bACheckWrappConv:=TRUE;
ELSE bACheckWrappConv:=FALSE; END_IF


						(*######################     Cone 1 Alignment checking####################*)

IF bQAWrappingConveyorMotor1 AND b2_4SetHmiSelected AND  NOT bAPauseSeq THEN TON_3_24(IN:=TRUE , PT:= t#7s, Q=> , ET=> );  ELSE  TON_3_24(IN:=FALSE); END_IF

IF bAutoModeOn AND TON_3_24.Q AND NOT bIWrappingCone1  AND b2_4SetHmiSelected THEN
bAConeMissErrorAtWrpConvTemp1_24:=TRUE;
 END_IF

IF bAutoModeOn  AND bIWrappingCone1  AND b2_4SetHmiSelected THEN
bAConeMissErrorAtWrpConvTemp1_24:=FALSE;
 END_IF

IF bErrorReset THEN TON_3_24(IN:=FALSE); bAConeMissErrorAtWrpConvTemp1_24:=FALSE; END_IF

IF NOT bIEmergencySwitch OR bStopHmi  OR bServoOff OR bIMcStop THEN
bAConeMissErrorAtWrpConvTemp1_24:=FALSE;
 TON_3_24(IN:=FALSE);
TON_13_24(in:=FALSE);
ConeMissAlarm:='';
END_IF

						(*######################     Cone 1,2 ,3 Alignment checking####################*)


IF bWrapConvStopped2 AND b2_4SetHmiSelected AND  NOT bAPauseSeq THEN TON_4_24(IN:=TRUE , PT:= t#5s, Q=> , ET=> );  ELSE  TON_4_24(IN:=FALSE); END_IF


IF bAutoModeOn  AND  TON_4_24.Q AND  (NOT bIWrappingCone1 OR NOT bIWrappingCone2 OR NOT bIWrappingCone3 ) AND NOT bWrapConvStopped1_24exp
AND b2_4SetHmiSelected  THEN bAConeMissErrorAtWrpConvTemp2_24:=TRUE;
ELSE
 IF  bAutoModeOn AND b2_4SetHmiSelected AND bWrapConvStopped2   AND bIWrappingCone1 AND bIWrappingCone2 AND bIWrappingCone3 THEN
  TON_12_24(IN:=TRUE , PT:= t#0.7s, Q=> , ET=> );  TON_4_24(IN:=FALSE);

IF TON_12_24.Q AND b2_4SetHmiSelected THEN  bWrapConvStopped2:=FALSE; END_IF
 END_IF  END_IF


IF bErrorReset  AND bAConeMissErrorAtWrpConvTemp2_24 AND  bIWrappingCone1 AND bIWrappingCone2 AND bIWrappingCone3
 THEN TON_4_24(IN:=FALSE); TON_12_24(in:=FALSE); bAConeMissErrorAtWrpConvTemp2_24:=FALSE; ConeMissAlarm:=''; END_IF

IF NOT bIEmergencySwitch OR bStopHmi  OR bServoOff OR bIMcStop THEN
bAConeMissErrorAtWrpConvTemp2_24:=FALSE;
bWrapConvStopped2:=FALSE;
 TON_4_24(IN:=FALSE);
TON_12_24(in:=FALSE);
ConeMissAlarm:='';
END_IF



					(*######################     Cone 4  Alignment checking####################*)



IF bWrapConvStopped4_24exp AND b2_4SetHmiSelected  AND  NOT bAPauseSeq THEN TON_5_24(IN:=TRUE , PT:= t#5s, Q=> , ET=> );  ELSE  TON_5_24(IN:=FALSE); END_IF

IF  bAutoModeOn AND TON_5_24.Q AND NOT bIWrappingCone3 AND b2_4SetHmiSelected  THEN
 bAConeMissErrorAtWrpConvTemp3_24:=TRUE;
ELSE
IF bAutoModeOn  AND bIWrappingCone3 AND bWrapConvStopped4_24exp AND b2_4SetHmiSelected THEN
TON_11_24(IN:=TRUE , PT:= t#1s, Q=> , ET=> ); TON_5_24(IN:=FALSE);
IF  TON_11_24.Q THEN bWrapConvStopped4_24exp:=FALSE; END_IF
 END_IF   END_IF

IF bErrorReset AND bAConeMissErrorAtWrpConvTemp3_24 AND bIWrappingCone3 THEN
TON_5_24(IN:=FALSE); TON_11_24(in:=FALSE); bAConeMissErrorAtWrpConvTemp3_24:=FALSE; ConeMissAlarm:='';END_IF

IF NOT bIEmergencySwitch OR bStopHmi  OR bServoOff OR bIMcStop THEN
bAConeMissErrorAtWrpConvTemp3_24:=FALSE;
bWrapConvStopped4_24exp:=FALSE;
 TON_5_24(IN:=FALSE);
TON_11_24(in:=FALSE);
ConeMissAlarm:='';
END_IF


						(*######################     Cone 5, 6  Alignment checking####################*)



IF bWrapConvStopped3_24  AND b2_4SetHmiSelected  AND  NOT bAPauseSeq THEN TON_6_24(IN:=TRUE , PT:= t#5s, Q=> , ET=> );  ELSE  TON_6_24(IN:=FALSE); END_IF


IF bAutoModeOn AND b2_4SetHmiSelected AND  TON_6_24.Q AND ( NOT bIWrappingCone2 OR NOT bIWrappingCone3 ) THEN
 bAConeMissErrorAtWrpConvTemp4_24:=TRUE;
ELSE
IF bAutoModeOn AND b2_4SetHmiSelected AND   bIWrappingCone2 AND bIWrappingCone3 AND bWrapConvStopped3_24 THEN
TON_10_24(IN:=TRUE , PT:= t#2s, Q=> , ET=> );
IF TON_10_24.Q THEN  bWrapConvStopped3_24:=FALSE; END_IF
 END_IF    END_IF


IF bErrorReset  AND bAConeMissErrorAtWrpConvTemp4_24 AND bIWrappingCone2 AND bIWrappingCone3 THEN
 TON_6_24(IN:=FALSE) ;  TON_10_24(in:=FALSE); bAConeMissErrorAtWrpConvTemp4_24:=FALSE; ConeMissAlarm:='';END_IF


IF NOT bIEmergencySwitch OR bStopHmi  OR bServoOff OR bIMcStop THEN
bAConeMissErrorAtWrpConvTemp4_24:=FALSE;
bWrapConvStopped3_24:=FALSE;
 TON_6_24(IN:=FALSE);
TON_10_24(in:=FALSE);
ConeMissAlarm:='';
END_IF



						(*######################     Cone 7, 8  Alignment checking####################*)




IF bWrapConvStopped4_24  AND b2_4SetHmiSelected  AND  NOT bAPauseSeq THEN TON_8_24(IN:=TRUE , PT:= t#5s, Q=> , ET=> );  ELSE  TON_8_24(IN:=FALSE); END_IF

IF TON_8_24.Q AND b2_4SetHmiSelected AND  bAutoModeOn  AND ( NOT bIWrappingCone2 OR NOT bIWrappingCone3 ) THEN
 bAConeMissErrorAtWrpConvTemp5_24:=TRUE;
ELSE
IF bAutoModeOn AND b2_4SetHmiSelected  AND  bIWrappingCone2 AND  bIWrappingCone3 AND bWrapConvStopped4_24    THEN
TON_9_24(IN:=TRUE , PT:= t#2s, Q=> , ET=> );
 IF TON_9_24.Q THEN bWrapConvStopped4_24:=FALSE; END_IF
  END_IF END_IF

IF bErrorReset AND bAConeMissErrorAtWrpConvTemp5_24 AND bIWrappingCone2 AND bIWrappingCone3    THEN
TON_8_24(IN:=FALSE); TON_9_24(in:=FALSE);   bAConeMissErrorAtWrpConvTemp5_24:=FALSE; ConeMissAlarm:='';END_IF

IF NOT bIEmergencySwitch OR bStopHmi  OR bServoOff OR bIMcStop THEN
bAConeMissErrorAtWrpConvTemp5_24:=FALSE;
bWrapConvStopped4_24:=FALSE;
 TON_8_24(IN:=FALSE);
TON_9_24(in:=FALSE);
ConeMissAlarm:='';
END_IF



(*============Wrapping Cone Missing Msg to Hmi=============*)

IF bAConeMissErrorAtWrpConvTemp1_24 AND b2_4SetHmiSelected THEN
ConeMissAlarm:='Allign the Cone  on Wrapping Conveyer ';

ELSIF bAConeMissErrorAtWrpConvTemp2_24 AND b2_4SetHmiSelected  THEN
ConeMissAlarm:='Allign the Cone  on Wrapping Conveyer ';

ELSIF bAConeMissErrorAtWrpConvTemp3_24  AND b2_4SetHmiSelected THEN
ConeMissAlarm:='Allign the Cone  on Wrapping Conveyer ';

ELSIF bAConeMissErrorAtWrpConvTemp4_24 AND b2_4SetHmiSelected  THEN
ConeMissAlarm:='Allign the Cone  on Wrapping Conveyer ';

ELSIF bAConeMissErrorAtWrpConvTemp5_24 AND b2_4SetHmiSelected  THEN
ConeMissAlarm:='Allign the Cone  on Wrapping Conveyer ';


ELSIF bACheckWrappConvError1 AND b2_4SetHmiSelected  THEN
ConeMissAlarm:='Check Wrapping Sensor 1 & 2 & 3';

ELSIF bACheckWrappConvError2  AND b2_4SetHmiSelected THEN
ConeMissAlarm:='Check Wrapping Sensor  1& 2 & 3';

ELSIF bACheckWrappConvError3 AND b2_4SetHmiSelected THEN
ConeMissAlarm:='Check Wrapping Sensor 1 & 2 & 3';

ELSIF bACheckWrappConvError4 AND b2_4SetHmiSelected THEN
ConeMissAlarm:='Check Wrapping Sensor  1& 2 & 3';

ELSIF bACheckWrappConvError5 AND b2_4SetHmiSelected THEN
ConeMissAlarm:='Check Wrapping Sensor  1& 2 & 3';


ELSIF NOT bAConeMissErrorAtWrpConvTemp1_24  AND NOT bAConeMissErrorAtWrpConvTemp2_24 AND NOT  bAConeMissErrorAtWrpConvTemp3_24
AND NOT bAConeMissErrorAtWrpConvTemp4_24 AND NOT bAConeMissErrorAtWrpConvTemp5_24 AND b2_4SetHmiSelected
AND NOT  bACheckWrappConvError1 AND NOT bACheckWrappConvError2 AND NOT bACheckWrappConvError3 AND NOT bACheckWrappConvError4
AND NOT bACheckWrappConvError5 THEN
ConeMissAlarm:='   ';
END_IF


END_IF
END_PROGRAM

(* POU New Folder/Cylinder_Alarm, ST *)
PROGRAM Cylinder_Alarm
VAR
	RS_Error_1:RS_Error;
	RS_Error_2:RS_Error;
	RS_Error_3:RS_Error;
	RS_Error_4:RS_Error;
	RS_Error_5:RS_Error;
	RS_Error_6:RS_Error;
	RS_Error_7:RS_Error;
	RS_Error_8:RS_Error;
	RS_Error_9:RS_Error;
	RS_Error_10:RS_Error;
	RS_Error_11:RS_Error;
	RS_Error_12:RS_Error;
	RS_Error_13:RS_Error;
	RS_Error_14:RS_Error;
	RS_Error_15:RS_Error;
	RS_Error_16:RS_Error;
	RS_Error_17:RS_Error;
	RS_Error_18:RS_Error;
	RS_Error_19:RS_Error;
	RS_Error_20:RS_Error;
	RS_Error_21:RS_Error;
	RS_Error_22:RS_Error;
	R_TRIG_2: R_TRIG;

	TestBool: BOOL;
	testIn: BOOL;
	ColoumConeSenError: RS_Error;
	SeparatorVerticalCylHomeRsErro: RS_Error;
	RS_Error_23: RS_Error;
	RS_Error_24: RS_Error;
	RS_Error_25: RS_Error;
	SupplyPressureError: RS_Error;
	BlinkTimer1: TON;
	BlinkTimer2: TON;
	BuzzerStopDly: TON;
	bEnableAlarm: BOOL;
	EmptyCartonDetect: RS_Error;
	TON_4: TON;
	bAConeMissErrorAtWrapConveyor: BOOL;
	BlinkTimer3: TON;
	BlinkTimer4: TON;
END_VAR
IF bASealBottomRsError OR SealTopBottomRsError OR bASealSepaX_axisRsError OR bASealSepaY_axisRsError  OR bAPolythinSheetError
OR bACartonOnGrossWtConv  OR bSealConveyerConePresent THEN
SealingUnitAlert:=TRUE;
ELSE SealingUnitAlert:=FALSE; END_IF

IF  bASupplyPressureError OR  SeparatorAlertbit  OR bGrossWieghtNOk OR SealBitAlert  OR  bQSealBitAlert (*OR bQSealBitAlert_24*)  OR bCartonFullDetectbit
OR bAConeMissErrorAtWrapConveyor OR baConePtrsentAtWrapConv  OR bHmiColourChangeBit2_24 OR bHmiColourChangeBit2 THEN
 PressureSeparatorAlert:=TRUE;
 ELSE PressureSeparatorAlert:=FALSE;END_IF

IF bAConeFeddCylFwdRsError OR bAWrap_PistRsError OR bAForwPistRsError OR bATiltPistRsError OR bAReversPistnRsError OR bEmptyCartonDetectError
THEN  PistonAlertAlarm:=TRUE;
ELSE PistonAlertAlarm:=FALSE; END_IF

IF bAColumnPushPistnRsError OR bAConeEjectPistnRsError OR bASepaHoriForwdEndRsError OR bSeparatorVerticalPistonEndRsSensed
OR bASepaVerCylhomeRsError OR bASepaHoriRevValveRsError THEN
GripperUnitAlert:=TRUE;
 ELSE GripperUnitAlert:=FALSE; END_IF

IF bASepaHoriRevValveRsError OR bAL_BTightHomeSenRsError OR bAGrossWtSenRsError OR bAGrossWtHomeSenRsError
OR bACartonSenRsError OR bARowStoppHomeSenRsError OR bAConeMissAtMatricConv THEN
 GrossWeightAlert:=TRUE;
ELSE GrossWeightAlert:=FALSE;END_IF

IF ERROR_ALERT AND NOT BlinkTimer1.Q THEN
 bEnableAlarm:=TRUE; ELSE bEnableAlarm:=FALSE;END_IF

IF SealingUnitAlert OR PressureSeparatorAlert OR PistonAlertAlarm OR GripperUnitAlert OR GrossWeightAlert (*AND NOT bANo_ErrorBit  *) OR bServoNotReady THEN
 ERROR_ALERT:=TRUE; sMianAlarmStatus:='Alarm Occured Go to Active Alarms'; ELSE ERROR_ALERT:=FALSE;sMianAlarmStatus:='No Alarms';END_IF
BlinkTimer1(IN:=(ERROR_ALERT AND NOT BlinkTimer2.Q) , PT:= t#0.5s, Q=> , ET=> );
BlinkTimer2(IN:= BlinkTimer1.Q, PT:=t#1.3s , Q=> , ET=> );(*
BuzzerStopDly(IN:= ERROR_ALERT, PT:=t#10s , Q=> , ET=> );  *)

BlinkTimer3(IN:= (bAEmergencyPressed AND NOT BlinkTimer4.Q) , PT:= t#0.5s, Q=> , ET=> );
BlinkTimer4(IN:= BlinkTimer3.Q, PT:=t#1.3s , Q=> , ET=> );

IF bAConeMissErrorAtWrpConv OR bConeMiss2AtWrapConv  OR
bACheckWrappConvError1_23 OR bACheckWrappConvError2 OR bACheckWrappConvError3 OR bACheckWrappConvError4  OR bACheckWrappConvError5  THEN
bAConeMissErrorAtWrapConveyor :=TRUE;
ELSE
bAConeMissErrorAtWrapConveyor:=FALSE; END_IF


IF ERROR_ALERT OR bAPauseSeq AND NOT bAMainIntStarted AND  bIEmergencySwitch  THEN bQATLAmber:=TRUE; bQATLGreen:=FALSE;  ELSE bQATLAmber:=FALSE; END_IF
IF BlinkTimer1.Q OR BlinkTimer3.Q   THEN  bQABuzzer:=TRUE; ELSE bQABuzzer:=FALSE; END_IF

(*===========Supply Prssure===========*)


SupplyPressureError(
	bValveOutOn:= (bManualModeOn OR bAutoModeOn)  (*TestBool*),                                    (*Change*)
	bReedSwithIn:=  bIPressureSwitch (* testIn*) ,
	bErroReset:=((* bErrorReset OR bANo_ErrorBit),*) bIPressureSwitch),
	sMsgIn:= ,
	RS_ErrChkDly:=t#10s ,
	bRsError=>bASupplyPressureError ,
	sMsgOut=> );

IF SupplyPressureError.bRsError THEN
SupplyPressureError.sMsgIn:='Supply Pressure NOT  OK' ;
ELSE
SupplyPressureError.sMsgIn:='Continue Machine Operation' ;
END_IF
sSupplyPressuremsg:=SupplyPressureError.sMsgIn;





(*......................................Cone Feeding Piston Alarm.............................*)


RS_Error_1(
	bValveOutOn:= bQAConeFeedingPistonValve  (*TestBool*),
	bReedSwithIn:=  bIConeFeedingPistonEnd (* testIn*) ,
	bErroReset:= ( bErrorReset OR bANo_ErrorBit),
	sMsgIn:= ,
	RS_ErrChkDly:=t#10s ,
	bRsError=>bAConeFeddCylFwdRsError ,
	sMsgOut=> );

IF RS_Error_1.bRsError THEN
RS_Error_1.sMsgIn:='Cone Feeding Piston End Sensor Timeout Error' ;
ELSE
RS_Error_1.sMsgIn:='Continue Machine Operation' ;
END_IF
HMIFeedPiston:=RS_Error_1.sMsgIn;


(*.......Wrapping  Piston Error Bit-----------------*)

IF bAWrap_1PistRsError OR bAWrap_2PistRsError OR bAWrap_3PistRsError THEN bAWrap_PistRsError:=TRUE;ELSE bAWrap_PistRsError:=FALSE; END_IF
(*IF bAWrap_PistRsError AND bErrorReset THEN bAWrap_PistRsError:=FALSE; END_IF*)

(*......................................Wrapping Channel Piston1 Alarm.............................*)


RS_Error_2(
	bValveOutOn:=bQAWrappingChannelPistonValve1,
	bReedSwithIn:=bIWrappingChannelPiston1_End,
	bErroReset:=( bErrorReset OR bANo_ErrorBit),
	sMsgIn:= ,
	RS_ErrChkDly:=t#10s ,
	bRsError=> bAWrap_1PistRsError,
	sMsgOut=> );
IF  RS_Error_2.bRsError  THEN
RS_Error_2.sMsgIn:=' Wrapping  Piston1 End Sensor Timeout Error' ;

ELSE
RS_Error_2.sMsgIn:='Continue Machine Operation' ;

END_IF

HMIWrapPiston1:=RS_Error_2.sMsgIn;

(*......................................Wrapping Channel Piston2 Alarm.............................*)

RS_Error_3(
	bValveOutOn:=bQAWrappingChannelPistonValve2,
	bReedSwithIn:=bIWrappingChannelPiston2_End,
	bErroReset:=( bErrorReset OR bANo_ErrorBit),
	sMsgIn:= ,
	RS_ErrChkDly:=t#10s ,
	bRsError=>bAWrap_2PistRsError ,
	sMsgOut=> );

IF  RS_Error_3.bRsError  THEN
RS_Error_3.sMsgIn:=' Wrapping  Piston2 End Sensor Timeout Error' ;


ELSE
RS_Error_3.sMsgIn:='Continue Machine Operation' ;
END_IF

HMIWrapPiston2:=RS_Error_3.sMsgIn;

(*......................................Wrapping Channel Piston3 Alarm.............................*)


RS_Error_4(
	bValveOutOn:=bQAWrappingChannelPistonValve3,
	bReedSwithIn:=bIWrappingChannelPiston3_End,
	bErroReset:=( bErrorReset OR bANo_ErrorBit),
	sMsgIn:= ,
	RS_ErrChkDly:=t#10s ,
	bRsError=>bAWrap_3PistRsError ,
	sMsgOut=> );

IF RS_Error_4.bRsError THEN
RS_Error_4.sMsgIn:=' Wrapping  Piston3 End Sensor Timeout Error' ;

ELSE
RS_Error_4.sMsgIn:='Continue Machine Operation' ;
END_IF

HMIWrapPiston3:=RS_Error_4.sMsgIn;



(*.................................Cone Forward Piston Alarm............................................*)

RS_Error_5(
	bValveOutOn:=bQAForwardPistonValve,
	bReedSwithIn:=bIForwardPistonEnd,
	bErroReset:=( bErrorReset OR bANo_ErrorBit),
	sMsgIn:= ,
	RS_ErrChkDly:=t#10s ,
	bRsError=>bAForwPistRsError ,
	sMsgOut=> );
IF  RS_Error_5.bRsError THEN
RS_Error_5.sMsgIn:=' Forward Piston End Sensor Timeout Error';
ELSE
RS_Error_5.sMsgIn:='Continue Machine Operation' ;
END_IF

HMIForwdPiston:=RS_Error_5.sMsgIn;




(*.................................Sealing Bottom Piston Alarm............................................*)

RS_Error_6(
	bValveOutOn:=bQASealingTopPistonValve,
	bReedSwithIn:=bISealingBottomPistonEnd,
	bErroReset:=( bErrorReset OR bANo_ErrorBit),
	sMsgIn:= ,
	RS_ErrChkDly:=t#10s ,
	bRsError=>bASealBottomRsError ,
	sMsgOut=> );
IF RS_Error_6.bRsError THEN
RS_Error_6.sMsgIn:='Sealing Bottom Piston End Sensor Timeout Error';
ELSE
RS_Error_6.sMsgIn:='Continue Machine Operation' ;
END_IF

HMISealBotPiston:=RS_Error_6.sMsgIn;

(*..............Top and Bottom Piston Error.....*)

IF bASealTopPistRsError OR bASealBottomRsError THEN SealTopBottomRsError:=TRUE; END_IF
IF SealTopBottomRsError AND bErrorReset THEN SealTopBottomRsError:=FALSE; END_IF


(*.................................Sealing Top Piston Alarm............................................*)

RS_Error_7(
	bValveOutOn:=bQASealingTopPistonValve,
	bReedSwithIn:=bISealingTopPistonEnd,
	bErroReset:=( bErrorReset OR bANo_ErrorBit),
	sMsgIn:= ,
	RS_ErrChkDly:=t#10s ,
	bRsError=>bASealTopPistRsError ,
	sMsgOut=> );
IF  RS_Error_7.bRsError THEN
RS_Error_7.sMsgIn:='Sealing Top Piston End Sensor Timeout Error';
ELSE
RS_Error_7.sMsgIn:='Continue Machine Operation' ;
END_IF

HMISealTopPiston:=RS_Error_7.sMsgIn;


(*.................................Sealing Seperator X Axis  Alarm............................................*)

RS_Error_8(
	bValveOutOn:=bQASealingSeparatorXAxisPistonValve,
	bReedSwithIn:=bISealingSeparatorXAxisEnd,
	bErroReset:=( bErrorReset OR bANo_ErrorBit),
	sMsgIn:= ,
	RS_ErrChkDly:=t#10s ,
	bRsError=>bASealSepaX_axisRsError ,
	sMsgOut=> );
IF RS_Error_8.bRsError THEN
RS_Error_8.sMsgIn:=' X- Axis Piston End Sensor Timeout Error';
ELSE
RS_Error_8.sMsgIn:='Continue Machine Operation' ;
END_IF
HmiXAxisPiston:=RS_Error_8.sMsgIn;

(*.................................Sealing Seperator Y Axis  Alarm...........................................*)

RS_Error_9(
	bValveOutOn:=bQASealingSeparatorYAxisPistonValve,
	bReedSwithIn:=bISealingSeparatorYAxisEnd,
	bErroReset:=( bErrorReset OR bANo_ErrorBit),
	sMsgIn:= ,
	RS_ErrChkDly:=t#10s ,
	bRsError=>bASealSepaY_axisRsError ,
	sMsgOut=> );
IF RS_Error_9.bRsError THEN
RS_Error_9.sMsgIn:=' Y-Axis Piston End Sensor Timeout Error';
ELSE
RS_Error_9.sMsgIn:='Continue Machine Operation' ;
END_IF
HmiYAxisPiston:=RS_Error_9.sMsgIn;

	(*----------------------Tilting Piston Error-----------------*)

	RS_Error_10(
		bValveOutOn:=bQAConeTiltingPistonValve,
		bReedSwithIn:=bITiltingEnd,
		bErroReset:=( bErrorReset OR bANo_ErrorBit),
		sMsgIn:= ,
		RS_ErrChkDly:=t#10s ,
		bRsError=>bATiltPistRsError ,
		sMsgOut=> );
	IF RS_Error_10.bRsError THEN
	RS_Error_10.sMsgIn:=' Tilting Piston End Sensor Timeout Error';
	ELSE
	RS_Error_10.sMsgIn:='Continue Machine Operation' ;
	END_IF
	HmiTiltPiston:=RS_Error_10.sMsgIn;


(*----------------------Reverse Piston Error-----------------*)

RS_Error_11(
	bValveOutOn:=bQAReversePistonValve,
	bReedSwithIn:=bIReversePistonEnd,
	bErroReset:=( bErrorReset OR bANo_ErrorBit),
	sMsgIn:= ,
	RS_ErrChkDly:=t#10s ,
	bRsError=>bAReversPistnRsError ,
	sMsgOut=> );
IF RS_Error_11.bRsError THEN
RS_Error_11.sMsgIn:=' Reverse Piston End Sensor Timeout Error';
ELSE
RS_Error_11.sMsgIn:='Continue Machine Operation' ;
END_IF
HmiReverPiston:=RS_Error_11.sMsgIn;

(*---------------------- Piston Error-----------------*)
(*
RS_Error_12(
	bValveOutOn:=bQReversePistonValve,
	bReedSwithIn:=bIReversePistonEnd,
	bErroReset:=bErrorReset ,
	sMsgIn:= ,
	RS_ErrChkDly:=t#20s ,
	bRsError=> ,
	sMsgOut=> );
IF RS_Error_12.bRsError THEN
RS_Error_12.sMsgIn:='Revese Piston End Sensor Timeout Error';
ELSE
RS_Error_12.sMsgIn:='Continue Machine Operation' ;
END_IF
HmiReverPiston:=RS_Error_12.sMsgIn;
*)

(*---------------------- Column X AxisPiston Error-----------------*)

RS_Error_13(
	bValveOutOn:=bQAColumnPushPistonValve,
	bReedSwithIn:=bIColumnPushPistonEnd,
	bErroReset:=( bErrorReset OR bANo_ErrorBit),
	sMsgIn:= ,
	RS_ErrChkDly:=t#10s ,
	bRsError=>bAColumnPushPistnRsError ,
	sMsgOut=> );
IF RS_Error_13.bRsError THEN
RS_Error_13.sMsgIn:=' Column Push Piston End Sensor Timeout Error';
ELSE
RS_Error_13.sMsgIn:='Continue Machine Operation' ;
END_IF
HmiColuPushrPiston:=RS_Error_13.sMsgIn;

(*---------------------- Cone Ejection End Piston Error-----------------

RS_Error_14(
	bValveOutOn:=bQAConeEjectionPistonValve,
	bReedSwithIn:=bIConeEjectionPistonHome,
	bErroReset:=bErrorReset ,
	sMsgIn:= ,
	RS_ErrChkDly:=t#10s ,
	bRsError=> bAConeEjectPistnRsError,
	sMsgOut=> );
IF RS_Error_14.bRsError THEN
RS_Error_14.sMsgIn:=' Cone Ejection Piston End Sensor Timeout Error';
ELSE
RS_Error_14.sMsgIn:='Continue Machine Operation' ;
END_IF
HmiConeEjePiston:=RS_Error_14.sMsgIn;*)

(*---------------------- Cone Ejection Home Piston Error-----------------*)
(*
RS_Error_15(
	bValveOutOn:=bQConeEjectionPistonValve,
	bReedSwithIn:=bIConeEjectionPistonHome,
	bErroReset:=bErrorReset ,
	sMsgIn:= ,
	RS_ErrChkDly:=t#20s ,
	bRsError=> ,
	sMsgOut=> );
IF RS_Error_15.bRsError THEN
RS_Error_15.sMsgIn:=' Cone Ejection Piston Home Sensor Timeout Error';
ELSE
RS_Error_15.sMsgIn:='Continue Machine Operation' ;
END_IF
HmiColuPushrPiston:=RS_Error_15.sMsgIn;

*)

(*---------------------- Separator Horizontal  Forward End Piston Error-----------------*)

RS_Error_16(
	bValveOutOn:=bQASeparatorHorizontalPistonValveFwd,
	bReedSwithIn:=bISeparatorHorizontalPistonHome,
	bErroReset:=( bErrorReset OR bANo_ErrorBit),
	sMsgIn:= ,
	RS_ErrChkDly:=t#15s ,
	bRsError=>bASepaHoriForwdEndRsError ,
	sMsgOut=> );
IF RS_Error_16.bRsError THEN
RS_Error_16.sMsgIn:=' Separator Horizontal Piston End Sensor Timeout Error';
ELSE
RS_Error_16.sMsgIn:='Continue Machine Operation' ;
END_IF
HmiSepHorizPiston:=RS_Error_16.sMsgIn;


(*---------------------- Separator Vertical End Piston Error-----------------*)

IF bAutoModeOn AND bASepVerticalCylEndRsErrChkBit AND R_TRIG_2.Q  THEN bSeparatorVerticalPistonEndRsSensed:=TRUE; END_IF
R_TRIG_2(CLK:= bISeparatorVerticalPistonEnd , Q=> );


RS_Error_17(
	bValveOutOn:=bASepVerticalCylEndRsErrChkBit,
	bReedSwithIn:=bSeparatorVerticalPistonEndRsSensed,
	bErroReset:=( bErrorReset OR bANo_ErrorBit),
	sMsgIn:= ,
	RS_ErrChkDly:=t#5s ,
	bRsError=>bASepaVertiEndPistnRsError ,
	sMsgOut=> );
IF RS_Error_17.bRsError THEN
RS_Error_17.sMsgIn:=' Separator Vertical Piston End Sensor Timeout Error';
ELSE
RS_Error_17.sMsgIn:='Continue Machine Operation' ;
END_IF
HmiSepVertiPiston:=RS_Error_17.sMsgIn;

(*==========================Separator Vertical Cyl Hmoe Rs Error=======================*)
SeparatorVerticalCylHomeRsErro(
	bValveOutOn:=bASepVerticalCylRevRsErrChkBit,
	bReedSwithIn:=bISeparatorVerticalPistonHome,
	bErroReset:=( bErrorReset OR bANo_ErrorBit),
	sMsgIn:= ,
	RS_ErrChkDly:=t#10s ,
	bRsError=>bASepaVerCylhomeRsError ,
	sMsgOut=> );
IF SeparatorVerticalCylHomeRsErro.bRsError THEN
SeparatorVerticalCylHomeRsErro.sMsgIn:=' Separator Vertical Piston End Sensor Timeout Error';
ELSE
SeparatorVerticalCylHomeRsErro.sMsgIn:='Continue Machine Operation' ;
END_IF
HmiSepVeticCylHomeRsError:=SeparatorVerticalCylHomeRsErro.sMsgIn;





(*---------------------- Separator Horizontal Rev Rs Error-----------------*)

RS_Error_18(
	bValveOutOn:=bQASeparatorHorizontalPistonValveRev,
	bReedSwithIn:=bISeparatorHorizontalPistonEnd,
	bErroReset:=( bErrorReset OR bANo_ErrorBit),
	sMsgIn:= ,
	RS_ErrChkDly:=t#15s ,
	bRsError=>bASepaHoriRevValveRsError ,
	sMsgOut=> );
IF RS_Error_18.bRsError THEN
RS_Error_18.sMsgIn:=' Separator Hori. Reverse Piston End Sensor Timeout Error';
ELSE
RS_Error_18.sMsgIn:='Continue Machine Operation' ;
END_IF
HmiSepHoriRevPiston:=RS_Error_18.sMsgIn;


(*---------------------- Lenght Tight Home Sensor Error-----------------*)

RS_Error_19(
	bValveOutOn:=(bAServoDownDone AND NOT bAPauseSeq) ,
	bReedSwithIn:= (bILengthTightPistonHome AND  bIBreadthTightPistonHome) ,
	bErroReset:=( bErrorReset OR bANo_ErrorBit),
	sMsgIn:= ,
	RS_ErrChkDly:=t#10s ,
	bRsError=>bAL_BTightHomeSenRsError ,
	sMsgOut=> );
IF RS_Error_19.bRsError THEN
RS_Error_19.sMsgIn:=' Lenght Tight  Piston Home Sensor Timeout Error';
ELSE
RS_Error_19.sMsgIn:='Continue Machine Operation' ;
END_IF
HmiLengthPiston:=RS_Error_19.sMsgIn;


(*---------------------- Breadth Tight Home Sensor Error-----------------*)
(*
RS_Error_20(
	bValveOutOn:=bQABreadthTightPistonValve,
	bReedSwithIn:=bIBreadthTightPistonHome,
	bErroReset:=bErrorReset ,
	sMsgIn:= ,
	RS_ErrChkDly:=t#10s ,
	bRsError=> bABreadthTightHomeSenRsError,
	sMsgOut=> );
IF RS_Error_20.bRsError THEN
RS_Error_20.sMsgIn:=' Breadth  Tight  Piston Home Sensor Timeout Error';
ELSE
RS_Error_20.sMsgIn:='Continue Machine Operation' ;
END_IF
HmiBreadthPiston:=RS_Error_20.sMsgIn;
*)

(*---------------------- Gross Weight  End Sensor Error-----------------*)

RS_Error_21(
	bValveOutOn:=bQAGrossWtPiston,
	bReedSwithIn:=bIGrossWtPistonEnd,
	bErroReset:=( bErrorReset OR bANo_ErrorBit),
	sMsgIn:= ,
	RS_ErrChkDly:=t#10s ,
	bRsError=>bAGrossWtSenRsError ,
	sMsgOut=> );
IF RS_Error_21.bRsError THEN
RS_Error_21.sMsgIn:=' Gross Weight  Piston End Sensor Timeout Error';
ELSE
RS_Error_21.sMsgIn:='Continue Machine Operation' ;
END_IF
HmiGrossWtPiston:=RS_Error_21.sMsgIn;

(*===============================Gross wt Home Sensor Error=============*)



RS_Error_23(
	bValveOutOn:=GrossWtReedSwBit,
	bReedSwithIn:=bIGrossWtPistonHome,
	bErroReset:=( bErrorReset OR bANo_ErrorBit),
	sMsgIn:= ,
	RS_ErrChkDly:=t#5s ,
	bRsError=>bAGrossWtHomeSenRsError ,
	sMsgOut=> );
IF RS_Error_23.bRsError THEN
RS_Error_23.sMsgIn:=' Gross Weight  Piston End Sensor Timeout Error';
ELSE
RS_Error_23.sMsgIn:='Continue Machine Operation' ;
END_IF
HmiGrossWtHomePiston:=RS_Error_23.sMsgIn;




(*---------------------- Empty Carton Feeding Sensor Error-----------------*)

RS_Error_22(
	bValveOutOn:=bQACartonFeedingPistonValve,
	bReedSwithIn:=bICartonFeedingPistonEnd,
	bErroReset:=( bErrorReset OR bANo_ErrorBit),
	sMsgIn:= ,
	RS_ErrChkDly:=t#10s ,
	bRsError=>bACartonSenRsError ,
	sMsgOut=> );
IF RS_Error_22.bRsError THEN
RS_Error_22.sMsgIn:=' Empty Carton Feeding  Piston End Sensor Timeout Error';
ELSE
RS_Error_22.sMsgIn:='Continue Machine Operation' ;
END_IF
HmiEmptyCartonPiston:=RS_Error_22.sMsgIn;



ColoumConeSenError(
	bValveOutOn:=bA3COneCrossed,
	bReedSwithIn:=bIColumnconeDetection,
	bErroReset:=( bErrorReset OR bANo_ErrorBit),
	sMsgIn:= ,
	RS_ErrChkDly:=t#5s ,
	bRsError=>bAColoumnConeSenError ,
	sMsgOut=> );
IF ColoumConeSenError.bRsError THEN
ColoumConeSenError.sMsgIn:=' Column Cone Sensor Timeout Error';
ELSE
ColoumConeSenError.sMsgIn:='Continue Machine Operation' ;
END_IF
HmiColoumConeSen:=ColoumConeSenError.sMsgIn;

(*Change*)

(*---------------------- Row Stopper Home  Sensor Error-----------------*)

RS_Error_24(
	bValveOutOn:=bQARowStopperMotorRev1,
	bReedSwithIn:=bIRowStopperHome,
	bErroReset:=( bErrorReset OR bANo_ErrorBit),
	sMsgIn:= ,
	RS_ErrChkDly:=t#10s ,
	bRsError=>bARowStoppHomeSenRsError ,
	sMsgOut=> );
IF RS_Error_24.bRsError THEN
RS_Error_24.sMsgIn:=' Row Stopper Home Sensor Timeout Error';
ELSE
RS_Error_24.sMsgIn:='Continue Machine Operation' ;
END_IF
HmiEmptyCartonPiston:=RS_Error_24.sMsgIn;

(*==========Cone On Matrix Conveyor===========*)

IF bAConeOnMatrixConv THEN
HmiConeOnMatxConvey:='Clear the Cone from Matrix Conveyor';
ELSIF  NOT bAConeOnMatrixConv THEN HmiConeOnMatxConvey:='';
END_IF


(*Sealing Cone Conveyor Reset Logic=======*)

IF bErrorReset THEN SealConeMiss:='Continue Machine Operation'; END_IF


(*=========POlythin Sheet Feeding Error=========*)
(*
RS_Error_25(
	bValveOutOn:=bAWrappingCone123OnAuto ,
	bReedSwithIn:= bAFilmLoadedCom,
	bErroReset:=bErrorReset ,
	sMsgIn:= ,
	RS_ErrChkDly:= t#10s,
	bRsError=>bAPolythinSheetError ,
	sMsgOut=> );

IF RS_Error_25.bRsError THEN
RS_Error_25.sMsgIn:=' Row Stopper Home Sensor Timeout Error';
ELSE
RS_Error_25.sMsgIn:='Continue Machine Operation' ;
END_IF
HmiPolyThinFeedErr:=RS_Error_25.sMsgIn;
*)
IF bAPolythinSheetError AND bErrorReset   THEN  bFilmErrClear:=TRUE; RS_Error_25.sMsgIn:='Continue Machine Operation' ;bAPolythinSheetError:=FALSE ;END_IF



 IF NOT bIEmergencySwitch OR bStopHmi OR bIMcStop OR bServoOff  THEN
  bASealBottomRsError:=FALSE; SealTopBottomRsError:=FALSE;  bASealSepaX_axisRsError:=FALSE; bASealSepaY_axisRsError :=FALSE; bAPolythinSheetError:=FALSE; bACartonOnGrossWtConv :=FALSE;
 bSealConveyerConePresent:=FALSE;
  bASupplyPressureError :=FALSE;  SeparatorAlertbit  :=FALSE; bGrossWieghtNOk :=FALSE; SealBitAlert  :=FALSE; bCartonFullDetectbit  :=FALSE; bAEmergencyPressed  :=FALSE;
 bAConeMissErrorAtWrapConveyor:=FALSE;
 bAConeFeddCylFwdRsError :=FALSE; bAWrap_PistRsError :=FALSE; bAForwPistRsError :=FALSE; bATiltPistRsError :=FALSE; bAReversPistnRsError :=FALSE; bEmptyCartonDetectError:=FALSE;

 bAColumnPushPistnRsError :=FALSE; bAConeEjectPistnRsError :=FALSE; bASepaHoriForwdEndRsError :=FALSE; bSeparatorVerticalPistonEndRsSensed :=FALSE; bASepaVerCylhomeRsError :=FALSE; bASepaHoriRevValveRsError :=FALSE;

 bASepaHoriRevValveRsError :=FALSE; bAL_BTightHomeSenRsError :=FALSE; bAGrossWtSenRsError :=FALSE; bAGrossWtHomeSenRsError :=FALSE; bACartonSenRsError :=FALSE; bARowStoppHomeSenRsError:=FALSE;
 bAConeMissAtMatricConv  :=FALSE;  bANo_ErrorBit:=TRUE;
END_IF

IF bQAEmptyCartonConveyorMotor1 THEN TON_4(IN:=TRUE , PT:= t#30s, Q=> , ET=> ); ELSE  TON_4(IN:=FALSE); END_IF

IF bAutoModeOn AND TON_4.Q AND NOT bIEmptyCartonDetectionSensor THEN bEmptyCartonDetectError:=TRUE; HMIEmptyCartonDetectErr:= ' Place Carton At Empty Carton Conveyor';  END_IF

IF bAutoModeOn AND  bIEmptyCartonDetectionSensor  AND bErrorReset THEN bEmptyCartonDetectError:=FALSE ; HMIEmptyCartonDetectErr:= ' Continue Machine Operation';  TON_4(IN:=FALSE); END_IF

(*================Emergency Alarm======================*)

IF NOT bIEmergencySwitch THEN bAEmergencyPressed:=TRUE; ELSE bAEmergencyPressed:=FALSE; END_IF

IF bAEmergencyPressed (*AND BlinkTimer1.Q *)THEN bEmPopUp:=TRUE; ELSE bEmPopUp:=FALSE; END_IF
END_PROGRAM

(* POU New Folder/ServoError, ST *)
PROGRAM ServoError
VAR
	RServoHomeRsError: RS_Error;
	bGripperVerticalEndSensed: BOOL;
	RServoEndRsError: RS_Error;
END_VAR
(*-=============Servo Home Sensor Error==================*)

RServoHomeRsError(
	bValveOutOn:=bAServoFwdStart ,
	bReedSwithIn:=bIGripperVerticalHome ,
	bErroReset:=bErrorReset ,
	sMsgIn:= ,
	RS_ErrChkDly:=T#17s ,
	bRsError=> ,
	sMsgOut=> );
IF RServoHomeRsError.bRsError THEN
RServoHomeRsError.sMsgIn:=' Servo Home Sensor Timeout Error';
ELSE
RServoHomeRsError.sMsgIn:='Continue Machine Operation' ;
END_IF
HmiServoHome:=RServoHomeRsError.sMsgIn;

(*-=============Servo END Sensor Error==================*)


IF bChkEndSensor AND statusword.10 AND bIGripperVerticalEnd THEN  bGripperVerticalEndSensed:=TRUE; ELSE bGripperVerticalEndSensed:=FALSE;  END_IF


RServoEndRsError(
	bValveOutOn:=bChkEndSensor ,
	bReedSwithIn:=bGripperVerticalEndSensed ,
	bErroReset:=bErrorReset ,
	sMsgIn:= ,
	RS_ErrChkDly:=T#10s ,
	bRsError=> , 
	sMsgOut=> );

IF RServoEndRsError.bRsError THEN
RServoEndRsError.sMsgIn:=' Servo End Sensor Timeout Error';
ELSE
RServoEndRsError.sMsgIn:='Continue Machine Operation' ;
END_IF
HmiServoHome:=RServoHomeRsError.sMsgIn;

IF NOT bIServoReady THEN
bServoNotReady:=TRUE;
sServoErrMsg:=' Servo Fault';
ELSE
bServoNotReady:=FALSE;
sServoErrMsg:='Continue Machine Operation';
END_IF
END_PROGRAM

(* POU New Folder/SeparatorAlarm, ST *)
PROGRAM SeparatorAlarm
VAR
	TON_1: TON;
END_VAR
(*===========Separator Unit*)


IF  NOT bISeparatorDetectionSensor AND NOT bServoOff   AND bAutoModeOn THEN
TON_1(IN:=TRUE , PT:= t#1s, Q=> , ET=> ); ELSE  TON_1(IN:=FALSE);
END_IF
IF TON_1.Q AND NOT bISeparatorDetectionSensor THEN
SeparatorAlertbit :=TRUE;
HMISeparatorPaperDetec:=' Put Separator  in Separator Table  ';
ELSE
HMISeparatorPaperDetec:='Separator Level OK';
END_IF
IF SeparatorAlertbit AND bErrorReset THEN HMISeparatorPaperDetec:='Separator Level OK'; SeparatorAlertbit:=FALSE; TON_1(IN:=FALSE);END_IF




(*=========Gross Weight NOT OK Alarm======*)


IF bGrossWieghtNOk THEN
GrossWtAlarm:=' Gross Weight  Low/ Over';
ELSE
GrossWtAlarm:='Continue Machine Operation';
END_IF
IF bGrossWieghtNOk AND bErrorReset THEN HMISeparatorPaperDetec:='Gross Weight OK'; bGrossWieghtNOk:=FALSE;END_IF
END_PROGRAM

(* POU Auto/Gripper/Servo_Pgm, ST *)
PROGRAM Servo_Pgm
VAR
	step: INT;
	bAReset: BOOL;


	check: BOOL;
	Timer1: TON;
	btest: BOOL;
END_VAR
CASE step OF

	0:	IF bAReset  OR bASrevoAutoHome OR bRServoHome1 OR bRServoHome OR bServoHomeHmi  AND bAutoModeOn THEN
		bAGoCounterAuto3:=FALSE;
		bARampDisableAuto3:=FALSE;
		bAServoHoming:=TRUE;
		bARampDisableAuto:=FALSE;
		bAServoStartAuto:=FALSE;
		bARampDisableAuto4:=FALSE;
		bAGoCounterAuto4:=FALSE;
		Timer1(IN:=FALSE);
		bServoStopHmi:=FALSE;
		step:=Step+1;
		END_IF

	1:	bARampDisableRst:=TRUE;
		bAGoCounterRst:=FALSE;
		step:=Step+1;

	2: 	step:=Step+1;

	3:	iASetCounteValRst:=65535;
		step:=Step+1;


	4:	bASetCounterRst:=TRUE;
		IF iACounterVal = iASetCounteValRst (*AND btest*) THEN
		step:=Step+1;
		END_IF

	5:	 bASetCounterRst:=FALSE;
		bAReset:=FALSE;
		Step:=Step+1;

	6:	iATargetCounteValRst:=0;
		Step:=Step+1;

	7:	iASetFequencyRst:=1300;
		bAGoCounterRst:=TRUE;
		Step:=Step+1;

	8:	bARampDisableRst:=FALSE;
		Step:=Step+1;



	9:	IF bIGripperVerticalHome THEN
		Step:=Step+1;
		ELSIF NOT bIGripperVerticalHome AND iACounterVal = 0 THEN
		 Step:=1;
		END_IF


	10:	bARampDisableRst:=TRUE;
		bAGoCounterRst:=FALSE;
		iASetCounteValRst:=0;
		Step:=Step+1;



	11:	bASetCounterRst:=TRUE;
			Timer1(IN:=FALSE);
		Step:=Step+1;

	12:	bASetCounterRst:=FALSE;
		bHomingDone:=TRUE;
		bRServoHome:=FALSE;
		bRServoHome1:=FALSE;

		Step:=Step+1;

	13:	Timer1(IN:=TRUE , PT:=t#2s , Q=> , ET=> );
		IF Timer1.Q THEN Step:=0; END_IF

END_CASE




IF bAReset THEN
bAServoStartAuto:=FALSE;
END_IF


IF  NOT bIEmergencySwitch OR bStopHmi OR bServoOff  OR bIMcStop THEN
Step:=0;
iASetFequencyRst:=0;
END_IF
END_PROGRAM

(* POU Manual/Manual, ST *)
PROGRAM Manual
VAR
	b_SHPistonValveREVOffHmi: BOOL;
	Timer1: TON;
	step: INT;
	bIManualSealingTemp: BOOL;
	bManualSealEnable: BOOL;
	bManualSealEnable2: BOOL;
END_VAR
(*=============MANUAL OPERATION============*)





(*=============UNIT-A LIFT CYL MANUAL OPERATION==========*)


	IF  bManualModeOn AND bUA_LiftCylOnHmi THEN	bQMUnitA_LiftPistonValve:=TRUE; END_IF
	IF bManualModeOn AND bUA_LiftCylOffHmi THEN	bQMUnitA_LiftPistonValve:=FALSE; END_IF




(*=============UNIT-BLIFT CYL MANUAL OPERATION==========*)


	IF bManualModeOn AND bUB_LiftCylOnHmi THEN	bQMUnitB_LiftPistonValve:=TRUE; END_IF
	IF bManualModeOn AND bUB_LiftCylOffHmi THEN	bQMUnitB_LiftPistonValve:=FALSE; END_IF




(*=============UNIT-A ROW STOPPER MOTOR FWD & REV==========*)


	IF  bManualModeOn AND  bUA_RowStopperMotorFwdOnHmi  AND NOT bIUnitA_RowStopperEnd    THEN	bQMUnitA_RowStopperMotorForward:=TRUE; ELSE   bQMUnitA_RowStopperMotorForward:=FALSE; END_IF
	IF  bManualModeOn AND   bIUnitA_RowStopperEnd THEN bQMUnitA_RowStopperMotorForward:=FALSE; END_IF




	IF bManualModeOn AND bUA_RowStopperMotorRevOnHmi AND NOT bIUnitA_RowStopperHome THEN	bQMUnitA_RowStopperMotorReverse:=TRUE; ELSE  bQMUnitA_RowStopperMotorReverse:=FALSE;  END_IF
	IF  bManualModeOn AND   bIUnitA_RowStopperHome THEN  bQMUnitA_RowStopperMotorReverse:=FALSE;  END_IF



(*=============UNIT-B ROW STOPPER MOTOR FWD & REV==========*)


	IF  bManualModeOn AND  bUB_RowStopperMotorFwdOnHmi AND NOT  bIUnitB_RowStopperEnd   THEN	bQMUnitB_RowStopperMotorForward:=TRUE; ELSE  	bQMUnitB_RowStopperMotorForward:=FALSE;   END_IF
	IF  bManualModeOn AND   bIUnitB_RowStopperEnd THEN bQMUnitB_RowStopperMotorForward:=FALSE; END_IF




	IF bManualModeOn AND bUB_RowStopperMotorRevOnHmi  AND NOT   bIUnitB_RowStopperHome   THEN 	bQMUnitB_RowStopperMotorReverse:=TRUE; ELSE  bQMUnitB_RowStopperMotorReverse:=FALSE;    END_IF
	IF  bManualModeOn AND   bIUnitB_RowStopperHome THEN  bQMUnitB_RowStopperMotorReverse:=FALSE;  END_IF






(*
	IF bUB_RowStopperMotorFwdOnHmi THEN	bQMUnitB_RowStopperMotorForward:=TRUE;
	 ELSE  bQMUnitB_RowStopperMotorForward:=FALSE; END_IF



	IF bUB_RowStopperMotorRevOnHmi THEN	bQMUnitB_RowStopperMotorReverse:=TRUE;
	 ELSE bQMUnitB_RowStopperMotorReverse:=FALSE;  END_IF

*)


(*============= FULL CARTON CONVEYOR OPERATION==========*)


	IF bManualModeOn AND bUC_FullCartonConvOnHmi THEN	bQMUnitC_FullCartonConveyor:=TRUE; END_IF
	IF bManualModeOn AND bUC_FullCartonConvOffHmi THEN	bQMUnitC_FullCartonConveyor:=FALSE; END_IF




(*=============UNIT-C LIFT CYL MANUAL OPERATION==========*)


	IF bManualModeOn AND bUC_LiftCylOnHmi THEN	bQMUnitC_LiftPistonValve:=TRUE; END_IF
	IF bManualModeOn AND bUC_LiftCylOffHmi THEN	bQMUnitC_LiftPistonValve:=FALSE; END_IF



(**************************CONE FEEDING OPERATION***************************)

	IF bManualModeOn AND bCFPistonOnHmi THEN bQMConeFeedingPistonValve:=TRUE; END_IF
	IF bManualModeOn AND bCFPistonOffHmi THEN bQMConeFeedingPistonValve:=FALSE;END_IF

(*=============FORWARD PISTON VALVE=================*)

	IF bManualModeOn AND bFPValveOnHmi  THEN bQMForwardPistonValve:=TRUE;END_IF
	IF bManualModeOn AND bFPValveOffHmi THEN bQMForwardPistonValve:=FALSE;END_IF

(*=================REVERSE PISTON VALVE=================*)

	IF bManualModeOn AND bRPValveOnHmi THEN  bQMReversePistonValve:=TRUE;END_IF
	IF bManualModeOn AND bRPValveOffHmi THEN  bQMReversePistonValve:=FALSE;END_IF

(*=================WRAPPING CHANNEL1=================*)

	IF bManualModeOn AND bWrappingCPV1OnHmi THEN bQMWrappingChannelPistonValve1:=TRUE;END_IF
	IF bManualModeOn AND bWrappingCPV1OffHmi THEN bQMWrappingChannelPistonValve1:=FALSE;END_IF


(*=================WRAPPING CHANNEL2=================*)

	IF bManualModeOn AND bWrappingCPV2OnHmi THEN bQMWrappingChannelPistonValve2:=TRUE;END_IF
	IF bManualModeOn AND bWrappingCPV2OffHmi THEN bQMWrappingChannelPistonValve2:=FALSE;END_IF

(*=================WRAPPING CHANNEL3=================*)

	IF bManualModeOn AND bWrappingCPV3OnHmi THEN bQMWrappingChannelPistonValve3:=TRUE;END_IF
	IF bManualModeOn AND bWrappingCPV3OffHmi THEN bQMWrappingChannelPistonValve3:=FALSE;END_IF

(*=================SEALING TOP PISTON=================*)

	IF bManualModeOn AND bSealingTopPVOnHmi THEN bQMSealingTopPistonValve:=TRUE;END_IF
	IF bManualModeOn AND bSealingTopPVOffHmi THEN bQMSealingTopPistonValve:=FALSE;END_IF

(*=================SEALING BOTTOM PISTON=================*)

	IF bManualModeOn AND bSealingBottomPVOnHmi	 THEN bQMSealingBottomPistonValve:=TRUE;END_IF
	IF bManualModeOn AND bSealingBottomPVOffHmi THEN bQMSealingBottomPistonValve:=FALSE;END_IF

(*=================FEEDING CONVEYOR MOTOR=================*)

	IF  bManualModeOn AND       bFCMotorOnHmi THEN bQMFeedingConveyorMotor:=TRUE;END_IF
	IF   bManualModeOn AND      bFCMotorOffHmi THEN bQMFeedingConveyorMotor:=FALSE;END_IF

(*=================WRAPPING CONVEYOR MOTOR=================*)

	IF bManualModeOn AND bWCMotorOnHmi THEN bQMWrappingConveyorMotor:=TRUE;END_IF
	IF bManualModeOn AND bWCMotorOffHmi THEN bQMWrappingConveyorMotor:=FALSE;END_IF

(*=================SEALING CONVEYOR MOTOR=================*)

	IF bManualModeOn AND bSCMotorOnHmi THEN bQMSealingConveyorMotor:=TRUE;END_IF
	IF bManualModeOn AND bSCMotorOffHmi THEN bQMSealingConveyorMotor:=FALSE;END_IF

(*=================MATRIX CONVEYOR MOTOR=================*)

	IF bManualModeOn AND bMCMotorOnHmi THEN bQMMatrixConveyorMotor:=TRUE;END_IF
	IF bManualModeOn AND bMCMotorOffHmi THEN bQMMatrixConveyorMotor:=FALSE;END_IF

(*=================FLIM ROLLER MOTOR1=================*)

	IF bManualModeOn AND bFRMotor1OnHmi THEN bQMFilmRollerMotor1:=TRUE;END_IF
	IF bManualModeOn AND bFRMotor1OffHmi THEN bQMFilmRollerMotor1:=FALSE;END_IF

(*=================FLIM ROLLER MOTOR2=================*)

	IF bManualModeOn AND bFRMotor2OnHmi THEN bQMFilmRollerMotor2:=TRUE;END_IF
	IF bManualModeOn AND bFRMotor2OffHmi THEN bQMFilmRollerMotor2:=FALSE;END_IF

(*=================FLIM ROLLER MOTOR3=================*)

	IF bManualModeOn AND bFRMotor3OnHmi THEN bQMFilmRollerMotor3:=TRUE;END_IF
	IF bManualModeOn AND bFRMotor3OffHmi THEN bQMFilmRollerMotor3:=FALSE;END_IF
(*=================ROW STOPPER  MOTOR FWD=================*)

	IF bManualModeOn AND bRSMotorForwardOnHmi  AND NOT bIRowStopper3  THEN  bQMRowStopperMotorForward:=TRUE; ELSE   bQMRowStopperMotorForward:=FALSE; END_IF


(*=================ROW STOPPER  MOTOR REV=================*)

	IF bManualModeOn AND bRSMotorRevOnHmi AND NOT bIRowStopperHome   THEN  bQMRowStopperMotorReverse:=TRUE; ELSE bQMRowStopperMotorReverse :=FALSE ; END_IF

(*=================COLUMN STOPPER  MOTOR FWD=================*)

	IF bManualModeOn AND bCSMotorFwdOnHmi AND  NOT bIColumnStopper3  THEN bQMColumnStopperMotorForward:=TRUE; ELSE bQMColumnStopperMotorForward:=FALSE; END_IF


(*=================COLUMN STOPPER  MOTOR REV====================*)

	IF bManualModeOn AND bCSMotorRevOnHmi AND NOT  bIColumnStopperHome   THEN bQMColumnStopperMotorReverse:=TRUE; ELSE bQMColumnStopperMotorReverse:=FALSE; END_IF

(*==============SEALING SEPARATOR YPISTON VALVE===================*)

	IF bManualModeOn AND bSSYAxisPistonValveOffHmi THEN  bQMSealingSeparatorYAxisPistonValve:=TRUE;END_IF
	IF bManualModeOn AND bSSYAxisPistonValveOnHmi THEN  bQMSealingSeparatorYAxisPistonValve:=FALSE;END_IF


(*================SEALING SEPARATOR XPISTON VALVE=================*)

	IF bManualModeOn AND bSSXAxisPistonValveOnHmi THEN  bQMSealingSeparatorXAxisPistonValve:=TRUE;END_IF
	IF bManualModeOn AND bSSXAxisPistonValveOffHmi THEN  bQMSealingSeparatorXAxisPistonValve:=FALSE;END_IF

(*====================CONE TILTING PISTON  VALVE=====================*)

	IF bManualModeOn AND bCTPistonValveOnHmi THEN  bQMConeTiltingPistonValve:=TRUE;END_IF
	IF bManualModeOn AND bCTPistonValveOffHmi   THEN  bQMConeTiltingPistonValve:=FALSE;END_IF


(*====================COLUMN PUSH PISTON X  VALVE=====================*)

	IF bManualModeOn AND bCPushPistonValveOnHmi THEN  bQMColumnPushPistonValve:=TRUE;END_IF
	IF bManualModeOn AND bCPushPistonValveOffHmi THEN  bQMColumnPushPistonValve:=FALSE;END_IF



(*====================COLUMN PUSH PISTON Y VALVE=====================*)

	IF bManualModeOn AND bCPushPistonValveYOnHmi THEN  bQMColumnPushPistonValveY:=TRUE;END_IF
	IF bManualModeOn AND bCPushPistonValveYOffHmi THEN  bQMColumnPushPistonValveY:=FALSE;END_IF



(*=============SEPARATOR HORIZONTAL  PISTON VALVE=================*)

	IF bManualModeOn AND bSHPistonValveOnHmi THEN  bQMSeparatorHorizontalPistonValveFwd:=TRUE;END_IF                                             (* ============FOR Separator horizontal output interchnged============*)
	IF bManualModeOn AND bISeparatorHorizontalPistonHome THEN  bQMSeparatorHorizontalPistonValveFwd:=FALSE;END_IF





(*=================== SEPERATOR HORIZONTAL  PISTON VALVE REV ======================*)

	IF bManualModeOn AND bSHPistonValveREVOnHmi THEN   bQMSeparatorHorizontalPistonValveRev:=TRUE;END_IF                                (* ============FOR Separator horizontal output interchnged============*)
	IF bManualModeOn AND bISeparatorHorizontalPistonEnd THEN   bQMSeparatorHorizontalPistonValveRev:=FALSE;END_IF





(*=============SEPARATOR VERTICAL  PISTON VALVE=================*)

	IF bManualModeOn AND bSVPistonValveOnHmi THEN  bQMSeparatorVerticalPistonValve:=TRUE;END_IF
	IF bManualModeOn AND bSVPistonValveOffHmi THEN  bQMSeparatorVerticalPistonValve:=FALSE;END_IF

(*================CARTON FEEDING  PISTON VALVE==================*)

	IF bManualModeOn AND bCPistonValveOnHmi THEN  bQMCartonFeedingPistonValve:=TRUE;END_IF
	IF bManualModeOn AND bCPistonValveOffHmi THEN  bQMCartonFeedingPistonValve:=FALSE;END_IF

(*================CONE EJECTION  PISTON VALVE===================*)

	IF bManualModeOn AND bCEPistonValveOnHmi THEN bQAConeEjectionPistonValve:=TRUE;END_IF
	IF bManualModeOn AND bCEPistonValveOffHmi THEN 	bQAConeEjectionPistonValve:=FALSE;END_IF

(*===============LENGTH TIGHT  PISTON VALVE====================*)

	IF bManualModeOn AND bGrippercCloseHmi THEN  bQMLengthTightPistonValve:=TRUE;END_IF
	IF bManualModeOn  AND 	bGripperOpenHmi THEN bQMLengthTightPistonValve:=FALSE; END_IF

(*===============BREADTH TIGHT PISTON VALVE====================*)

	IF bManualModeOn AND bGrippercCloseHmi THEN  bQMBreadthTightPistonValve:=TRUE;END_IF
	IF bManualModeOn  AND 	bGripperOpenHmi THEN bQMBreadthTightPistonValve:=FALSE; END_IF

(*===============EMPTY CARTON CONVEYOR MOTOR================*)

	IF bManualModeOn AND bECCMotorOnHmi THEN  bQMEmptyCartonConveyorMotor:=TRUE;END_IF
	IF bManualModeOn AND bECCMotorOffHmi THEN  bQMEmptyCartonConveyorMotor:=FALSE;END_IF
(*================== CARTON CONVEYOR MOTOR====================*)

	IF bManualModeOn AND bCCMotorOnHmi THEN  bQMCartonConveyorMotor:=TRUE;END_IF
	IF bManualModeOn AND bCCMotorOffHmi THEN  bQMCartonConveyorMotor:=FALSE;END_IF

(*=================== VACCUM PISTON VALVE ======================*)

	IF bManualModeOn AND bVPValveOnHmi THEN  bQMVacuumPistonValve:=TRUE;END_IF
	IF bManualModeOn AND bVPValveOffHmi THEN  bQMVacuumPistonValve:=FALSE;END_IF



(*=================== GROSS WEIGHT  PISTON VALVE ======================*)

	IF bManualModeOn AND bGWPistonOnHmi THEN  bQMGrossWtPiston:=TRUE;END_IF
	IF bManualModeOn AND bGWPistonOffHmi1 THEN  bQMGrossWtPiston:=FALSE;END_IF


(*=================== GROSS WEIGHT  PISTON VALVE ======================*)

	IF bManualModeOn AND bRCOnHmi THEN  bQMRollerConvMotor:=TRUE;END_IF
	IF bManualModeOn AND bRCOffHmi THEN  bQMRollerConvMotor:=FALSE;END_IF





(*======================manual Sealing Logic==========================*)

IF NOT  bAutoModeOn AND bIManualSealing THEN bManualSealEnable:=TRUE; ELSE bManualSealEnable:=FALSE; END_IF

IF   bAutoModeOn AND bAPauseSeq  AND bIManualSealing THEN bManualSealEnable2:=TRUE; ELSE bManualSealEnable2:=FALSE; END_IF

CASE step OF

	0:	IF  ( bManualSealEnable OR bManualSealEnable2  )THEN bMManualSealOn:=TRUE; step:=step+1;  END_IF

	1:	Timer1(IN:= FALSE);
		bQMSealingTopPistonValve:=TRUE;
		step:=step+1;

	2:	 IF bISealingBottomPistonEnd AND bISealingTopPistonEnd THEN
		 step:=step+1;
		END_IF

	3:	Timer1(IN:=TRUE , PT:=t#2s , Q=> , ET=> );
		IF Timer1.Q THEN step:=step+1; END_IF


	4:	bMManualSealOn:=FALSE;
		bQMSealingTopPistonValve:=FALSE;
		Timer1(IN:= FALSE);
		 step:=step+1;

	5:	step:=0;

END_CASE

IF NOT bIEmergencySwitch OR bIMcStop OR bServoOff OR  bStopHmi THEN

bQMUnitA_LiftPistonValve:=FALSE;
bQMUnitB_LiftPistonValve:=FALSE;
bQMUnitA_RowStopperMotorForward:=FALSE;
bQMUnitA_RowStopperMotorReverse:=FALSE;
bQMUnitB_RowStopperMotorForward:=FALSE;
bQMUnitB_RowStopperMotorReverse:=FALSE;
bQMUnitC_FullCartonConveyor:=FALSE;
bQMUnitC_LiftPistonValve:=FALSE;
bQMConeFeedingPistonValve:=FALSE;
bQMForwardPistonValve:=FALSE;
 bQMReversePistonValve:=FALSE;
 bQMWrappingChannelPistonValve1:=FALSE;
 bQMWrappingChannelPistonValve2:=FALSE;
 bQMWrappingChannelPistonValve3:=FALSE;
bQMSealingTopPistonValve:=FALSE;
bQMSealingBottomPistonValve:=FALSE;
 bQMFeedingConveyorMotor:=FALSE;
 bQMWrappingConveyorMotor:=FALSE;
bQMSealingConveyorMotor:=FALSE;
 bQMMatrixConveyorMotor:=FALSE;
 bQMFilmRollerMotor1:=FALSE;
 bQMFilmRollerMotor2:=FALSE;
 bQMFilmRollerMotor3:=FALSE;
bQMRowStopperMotorForward:=FALSE;
 bQMRowStopperMotorReverse :=FALSE ;
bQMColumnStopperMotorForward:=FALSE;
bQMSealingSeparatorYAxisPistonValve:=FALSE;
bQMSealingSeparatorXAxisPistonValve:=FALSE;
 bQMColumnPushPistonValve:=FALSE;
 bQMColumnPushPistonValveY:=FALSE;
bQMColumnPushPistonValveY:=FALSE;
 bQMSeparatorHorizontalPistonValveFwd:=FALSE;
 bQMSeparatorHorizontalPistonValveRev:=FALSE;
bQMSeparatorVerticalPistonValve:=FALSE;
bQMCartonFeedingPistonValve:=FALSE;
	(*bQAConeEjectionPistonValve:=FALSE;  *)
 bQMLengthTightPistonValve:=FALSE;
bQMBreadthTightPistonValve:=FALSE;
 bQMEmptyCartonConveyorMotor:=FALSE;
bQMCartonConveyorMotor:=FALSE;
 bQMVacuumPistonValve:=FALSE;
bQMGrossWtPiston:=FALSE;
 bQMRollerConvMotor:=FALSE;
bMManualSealOn:=FALSE;
bQMSealingTopPistonValve:=FALSE;
	step:=0;
END_IF
END_PROGRAM

(* POU Auto/Gripper/Jogging, ST *)
PROGRAM Jogging
VAR

	start: BOOL;
	bMonitor: BOOL;
	Timer1: TON;
	Timer3: TON;
	RT_JogMOde: R_TRIG;
	Start1: BOOL;
	JogStartTemp: BOOL;
	TON_1: TON;
	iTorqueActtemp: INT;
	MonitoBit: BOOL;
	MonitoBittemp: BOOL;
	jogFast: BOOL;
	testbit: BOOL;

	R_TRIG_2: R_TRIG;

	bServoFirstHome: BOOL;
	bJogNegative: BOOL;
END_VAR
VAR_INPUT
	Timer2: TON;
END_VAR
IF NOT bIEmergencySwitch OR  bStopHmi  OR bServoOff OR bIMcStop THEN
Timer3(IN:=FALSE);
iControlWord1:=7;
bAModeWrite:=FALSE;
start:=FALSE;
jogFast:=FALSE;
Timer1(IN:=FALSE);
Timer2(IN:=FALSE);
bServoOnCone:=FALSE;
bServoHome:=FALSE;
TON_1(IN:=FALSE);
JogStep:=0;
END_IF


(*=================Jog Mode Change Operation==================*)

R_TRIG_2(CLK:=bJogStart , Q=> );


CASE JogStep OF

	0:	IF R_TRIG_2.Q THEN
		JogStep:=JogStep+1;
		END_IF

	1:	JogStep:=JogStep+1;

	2:	bJogStart:=FALSE;
		iControlWord1:= 6;
		Timer3(IN:=FALSE);
		JogStep:=JogStep+1;

	3:	iControlWord1:=7; JogStep:=JogStep+1;
	(*	IF.1 THEN JogStep:=JogStep+1; END_IF *)

	4:	IF ModeACT=255THEN JogStep:=6;
		ELSIF  ModeACT<>255 THEN JogStep:=JogStep+1;
		END_IF

	5:	ModeWrite:=-1;
		JogStep:=JogStep+1;

	6:	bAModeWrite:=TRUE;
		Timer3(IN:=TRUE , PT:=T#100ms , Q=> , ET=> );
		IF Timer3.Q THEN JogStep:=JogStep+1;  END_IF

	7:	IF ModeACT=255THEN  iControlWord1:=15;  R_TRIG_2();  bAModeWrite:=FALSE;  JogStep:=0; END_IF



END_CASE

(*=========Jog Mode Bit==============*)



(*==============Jog Mode Operation Logic==============*)

start:=TRUE;

Timer1(IN:=(start AND NOT Timer2.Q)  , PT:=t#50ms , Q=> , ET=> );

Timer2(IN:=Timer1.Q , PT:=t#50ms , Q=> , ET=> );


bMonitor:=Timer1.Q;



IF  bJogNegativeHmi THEN  bJogNegative:=TRUE; ELSE bJogNegative:=FALSE; END_IF



JogModeVar.0:= (bJogNegative AND NOT bIGripperVerticalHome)  ;

JogModeVar.1:= ( bJogPositiveHmi AND NOT bIGripperVerticalEnd) ;

JogModeVar.2:= ( jogFast);

bJogWrite:= ( bMonitor AND NOT bAutoModeOn);

IF bManualModeOn THEN
jogFast:=TRUE;
ELSE
jogFast:=FALSE;
END_IF



IF bIGripperVerticalHome AND bAutoModeOn THEN bServoFirstHome:=FALSE; END_IF

(*============Cone hitting Error Logic====================*)

IF( bServoStartedInAuto AND ModeACT = 1  )    AND  rServiActPosHmi <= -570.00 AND   iControlWord1= 31 THEN


IF    iTorqAvg >0  AND  iTorqAvg <= 100 THEN   bServoOnCone:=TRUE;  END_IF

IF bServoOnCone THEN  iControlWord1:=0; (*TON_1(IN:=TRUE , PT:=t#50ms , Q=> , ET=> );*) bServoHome:=TRUE; ELSE  TON_1(IN:=FALSE);    END_IF
END_IF
END_PROGRAM

(* POU Auto/Gripper/ServoSetting, ST *)
PROGRAM ServoSetting
VAR

	PickDisplace: Scale;
	rPickPosMaxHmi: REAL := 760.00;
	rPickDisplaceOut: REAL;
	DropDisplace: Scale;
	rDropPosMinHmi: REAL;
	rDropPosMaxHmi: REAL;
	ScaleActPos: Scale;
	ActionStatus: ADSREAD;
	ServoActStatus: DINT;
	start: BOOL;
	Timer1: TON;
	Timer2: TON;
	bMonitor: BOOL;
	JogModeVarTemp1: BOOL;
	JogModeVarTemp2: BOOL;
	bJogWritetemp: BOOL;


(*===========AVg variable=====*)

	i: INT;
	j: INT;
	Arr_r1Load: ARRAY [0..99] OF INT;
	r1Sum_LoadVal: DINT;
	Arr_r2Load: ARRAY[0..99] OF REAL;
	r2Sum_LoadVal: LREAL;
	Arr_r3Load: ARRAY[0..99] OF REAL;
	r3Sum_LoadVal: LREAL;
	Arr_r4Load: ARRAY[0..99] OF REAL;
	r4Sum_LoadVal: LREAL;

	r1Sum_TorqVal: INT;
	R_TRIG_1: R_TRIG;
END_VAR
statusWord;
(*==========Servo Movement Scaling=================*)



PickDisplace(
	INPUT:=iPickPosHmi ,
	INPUTMIN:= 0.00,
	INPUTMAX:=750.00 ,
	OUTPUTMIN:=0.00 ,
	OUTPUTMAX:=28700.00 ,
	OUTPUT=>rTargetPos );

rTargetPosFinal:= REAL_TO_UINT(rTargetPos * -1);
rPickVeloFinal:=REAL_TO_UINT ( rPickVeloHmi);



DropDisplace(
	INPUT:=iDropPosHmi ,
	INPUTMIN:= 0,
	INPUTMAX:=750 ,
	OUTPUTMIN:=0 ,
	OUTPUTMAX:=28700 ,
	OUTPUT=>rDropPosFinal );


rDropVeloFinal:=rDropVeloHmi;


ScaleActPos(
	INPUT:=PosAct ,
	INPUTMIN:=0 ,
	INPUTMAX:=28700,
	OUTPUTMIN:=0 ,
	OUTPUTMAX:=750 ,
	OUTPUT=>rServiActPosHmi );
(*
ActionStatus(
	NETID:='5.34.251.157.3.1' ,
	PORT:=4097 ,
	IDXGRP:=16#310C ,
	IDXOFFS:= 8,
	LEN:= 4,
	DESTADDR:= (ADR(ServoActStatus)),
	READ:=bMonitor ,
	TMOUT:=default_ads_timeout ,
	BUSY=> ,
	ERR=> ,
	ERRID=> );

*)


(*===========Servo Status monitoring Blinker============*)

start:=TRUE;

Timer1(IN:=(start AND NOT Timer2.Q)  , PT:=t#10ms , Q=> , ET=> );

Timer2(IN:=Timer1.Q , PT:=t#10ms , Q=> , ET=> );


bMonitor:=Timer1.Q;



R_TRIG_1(CLK:=bMonitor , Q=> );


IF  R_TRIG_1.Q THEN
i:=i+1;
FOR j:=29 TO 1 BY -1 DO
Arr_r1Load[0]:= ReadActCur;
Arr_r1Load[j]:=Arr_r1Load[j-1];
END_FOR

END_IF


IF i>=29 THEN
FOR j:=0 TO 29 BY 1 DO
	r1Sum_LoadVal:=r1Sum_LoadVal+Arr_r1Load[j];
END_FOR
iTorqAvg:= DINT_TO_INT ((r1Sum_LoadVal/29));
	r1Sum_LoadVal:=0;
	i:=0;
END_IF
END_PROGRAM

(* POU StartUp/INT_All, ST *)
PROGRAM INT_All
VAR
	bCartonOnConv: BOOL;
	step: INT;
	TON_1: TON;
	TON_2: TON;
	TON_1Running: BOOL;
	bARCartanConvOnTemp: BOOL;
	R_TRIG_2: R_TRIG;
	bAOneMinConvReady2: BOOL;
	TON_3: TON;
	bAOneMinConvReady1: BOOL;
END_VAR
IF bInitializeHmi  AND bMCStartInAuto AND bAutoModeOn AND NOT bAinterlockinit  AND NOT bASupplyPressureError AND NOT bServoOff  AND NOT bIMcStop
AND NOT bStopHmi  THEN
	bAInitializeSeq:=TRUE;
	bAMainIntStarted:=TRUE;
	bAinterlockinit:=TRUE;
	 bANo_ErrorBit:=FALSE;
ELSE
	bAInitializeSeq:=FALSE;
END_IF

	R_TRIG_2(CLK:= bRowStopperIntOver  , Q=> );


IF NOT bIEmergencySwitch OR  R_TRIG_2.Q OR bServoOff  OR  bIMcStop OR bStopHmi  THEN bAMainIntStarted:=FALSE; END_IF
IF NOT bIEmergencySwitch OR  (*R_TRIG_2.Q OR*) bServoOff  OR  bIMcStop OR bStopHmi  THEN bAinterlockinit:=FALSE; END_IF
WrapConvRst();
SealingConvRst();
MatrixConvRst();
SealingUnitRst();


(*
AlarmList();
*)



(*=============FULL CARTON CONVEYOR INITIALIZE LOGIC==========*)



(*=============FULL CARTON CONVEYOR INITIALIZE LOGIC==========*)

	IF  bAIntStarted AND  (   bICartonPosition1 OR  bICartonPosition2 OR  bICartonPosition3 )    THEN bCartonOnConv:=TRUE;   END_IF

	IF bAInitializeSeq THEN bAIntStarted:=TRUE; END_IF
	IF 	bAIntStarted  AND  bCartonOnConv   AND bAutoModeOn  THEN
	bCartonFullDetectbit:=TRUE;
	sCartonConvStatus:='Clear the Cone on Carton Conveyor';
	ELSIF 	bAIntStarted AND NOT bCartonOnConv AND bAutoModeOn THEN
	bClearConeInt:=TRUE;
	bCartonOnConv:=FALSE;

	sCartonConvStatus:='';
	END_IF

	IF bCartonFullDetectbit AND bErrorReset THEN bCartonOnConv:=FALSE;  bCartonFullDetectbit:=FALSE; sCartonConvStatus:='Continue Machie Operation'; END_IF




CASE  step OF

	0:	IF bAInitializeSeq THEN TON_3(IN:=FALSE); TON_2(IN:=FALSE);
		 step:=step+1; END_IF
	1: 	bQROneMinConvStart:=TRUE;
		 step:=step+1;

	2:	TON_2(IN:= TRUE, PT:=t#10s , Q=> , ET=> );
		IF  TON_2.Q THEN step:=step+1; END_IF

	3:	IF bIGrossWtDeductSensor THEN bACartonOnGrossWtConv:=TRUE; sOneMinConMsg:=' Clear Cone At Gross Weight Conveyor'; bQROneMinConvStart:=FALSE;  step:=step+1;
		ELSIF NOT bIGrossWtDeductSensor THEN   step:=step+2;
		END_IF

	4: 	IF NOT  bIGrossWtDeductSensor AND bErrorReset THEN bACartonOnGrossWtConv:=FALSE;   sOneMinConMsg:='Continue Machine Operation'; step:=step+1; END_IF

	5:
		bQROneMinConvStart:=FALSE;
		bAOneMinConvReady1:=TRUE;
		 step:=step+1;

	6:	IF bOneMinConvOver THEN TON_3(IN:=FALSE); TON_2(IN:= FALSE); bAOneMinConvReady2:=TRUE;  step:=step+1; END_IF

	7:	bOneMinConvOver:=FALSE;
		TON_3(IN:=TRUE , PT:=t#2s , Q=> , ET=> );
		IF TON_3.Q THEN  step:=step+1; END_IF

	8:	TON_3(IN:=FALSE);
		 step:=6;

END_CASE

IF  bAOneMinConvReady1 OR  bAOneMinConvReady2 THEN bAOneMinConvReady:=TRUE;  bAOneMinConvReady1:=FALSE; bAOneMinConvReady2:=FALSE; END_IF




	IF bCartonFullDetectbit AND  bAutoModeOn THEN
	bHmiColourChangeBit:=TRUE;
HmiFullCartonAtConveyer:='Clear Carton  At Full Carton Conveyor';
ELSE
bHmiColourChangeBit:=FALSE;
HmiFullCartonAtConveyer:=' Continue Machine Operation';

END_IF


IF NOT bIEmergencySwitch OR bStopHmi OR bIMcStop OR bServoOff  THEN
bAOneMinConvReady1:=FALSE;
  bAOneMinConvReady2:=FALSE;
TON_3(IN:=FALSE);
bQROneMinConvStart:=FALSE;
bACartonOnGrossWtConv:=FALSE;
sOneMinConMsg:='Continue Machine Operation';
step:=0;
END_IF
END_PROGRAM

(* POU StartUp/WrapConvRst, ST *)
PROGRAM WrapConvRst
VAR
	step: INT;
	bConeAtWrppingConveyor1: BOOL;
	TON_1: TON;
	bConePresent: BOOL;
	bAResetHmitemp: BOOL;
	TON_1Running: BOOL;
	bConePresenttemp: BOOL;
END_VAR
CASE step OF

	0:	 IF bSealingUnitIntOver AND bAutoModeOn THEN
		bQAWrappingConveyorMotor1:=FALSE;
		bQAWrappingConveyorMotor2:=FALSE;
		bQAWrappingConveyorMotor3:=FALSE;
		bQAWrappingConveyorMotor4:=FALSE;
		bQAWrappingConveyorMotor5:=FALSE;
		bQAWrappingConveyorMotor3_23:=FALSE;
		bQAWrappingConveyorMotor4_23:=FALSE;
		TON_1(IN:=FALSE);
		step:=step+1;
		END_IF

	1:	bQRWrappingConveyorMotor:=TRUE;
		bSealingUnitIntOver:=FALSE;
		step:=step+1;

	2:	IF bConePresent THEN
		step:=step+2;
		ELSIF NOT bConePresent THEN
		step:=step+1;
		END_IF

	3:	IF  TON_1Running  AND bConePresent THEN
		step:=step+1;
		ELSIF TON_1.Q  AND NOT bConePresent THEN
		step:=step+2;
		END_IF

	4:	bQRWrappingConveyorMotor:=FALSE;
		TON_1(IN:=FALSE);
		sWrapConvStatus:='Clear Cone At Wapping Conveyor';
		baConePtrsentAtWrapConv:=TRUE;
		bConePresent:=FALSE;
		step:=step+1;

	5:	IF NOT bConePresent AND bAutoModeOn   THEN
		TON_1(IN:=FALSE);
		bQRWrappingConveyorMotor:=FALSE;
		sWrapConvStatus:=' ';
		baConePtrsentAtWrapConv:=FALSE;
		step:=step+1;
		END_IF

	6:	TON_1(IN:=FALSE);
		bWrpConvIntOver:=TRUE;
		step:=0;

END_CASE



IF TON_1.ET >t#1ms AND  TON_1.ET<=t#10s THEN
TON_1Running:=TRUE;
ELSE
TON_1Running:=FALSE;
END_IF



TON_1(IN:=bQRWrappingConveyorMotor , PT:=T#10s , Q=> , ET=> );






IF bIWrappingCone1 OR bIWrappingCone2 OR bIWrappingCone3 AND bQRWrappingConveyorMotor  THEN
bConePresent:=TRUE; ELSE bConePresent:=FALSE;
END_IF



IF baConePtrsentAtWrapConv THEN

sWrapConvStatus:='Clear Cone At Wapping Conveyor';
ELSE
sWrapConvStatus:='   ';
END_IF



IF NOT bIEmergencySwitch OR bStopHmi OR bIMcStop OR bServoOff THEN
		 bQAWrappingConveyorMotor1:=FALSE;
		bQAWrappingConveyorMotor2:=FALSE;
		bQAWrappingConveyorMotor3:=FALSE;
		bQAWrappingConveyorMotor4:=FALSE;
		bQAWrappingConveyorMotor5:=FALSE;
		bQAWrappingConveyorMotor3_23:=FALSE;
		bQAWrappingConveyorMotor4_23:=FALSE;
		bQRWrappingConveyorMotor:=FALSE;
		TON_1Running:=FALSE;
		baConePtrsentAtWrapConv:=FALSE;
		TON_1(IN:=FALSE);
		bWrpConvIntOver:=FALSE;
		bWrpConvIntOver:=FALSE;
		baConePtrsentAtWrapConv:=FALSE;
		step:=0;

END_IF
END_PROGRAM

(* POU StartUp/SealingConvRst, ST *)
PROGRAM SealingConvRst
VAR
	step: INT;
	bConeAtWrppingConveyor1: BOOL;
	TON_1: TON;
	bConePresent: BOOL;
	TON_1Running: BOOL;
END_VAR
IF NOT bIEmergencySwitch OR bStopHmi OR bIMcStop OR bServoOff  THEN
bQASealingConveyorMotor1:=FALSE;
		bQASealingConveyorMotor2:=FALSE;
		bQMSealingConveyorMotor:=FALSE;
		bQRSealingConveyorMotor:=FALSE;
		bConePresent:=FALSE;
		TON_1Running:=FALSE;
		sSealConvStatus:=' ';
		bSealConvIntOver:=FALSE;
		TON_1(IN:=FALSE);
		step:=0;
END_IF

CASE step OF

	0:	 IF bSealingUnitIntOver AND bAutoModeOn THEN
		bQASealingConveyorMotor1:=FALSE;
		bQASealingConveyorMotor2:=FALSE;
		bQMSealingConveyorMotor:=FALSE;
		step:=step+1;
		END_IF

	1:	bQRSealingConveyorMotor:=TRUE;
		bSealingUnitIntOver:=FALSE;
		step:=step+1;

	2:	IF bConePresent THEN
		step:=step+2;
		ELSIF NOT bConePresent THEN
		step:=step+1;
		END_IF

	3:	IF  TON_1Running  AND bConePresent THEN
		step:=step+1;
		ELSIF TON_1.Q  AND NOT bConePresent THEN
		step:=step+2;
		END_IF

	4:	bQRSealingConveyorMotor:=FALSE;
		TON_1(IN:=FALSE);
		bSealConveyerConePresent:=TRUE;
		sSealConvStatus:='Clear Cone At Sealing Conveyor';

		bConePresent:=FALSE;
		step:=step+1;

	5:	IF NOT bConePresent AND bAutoModeOn   THEN
		bSealConveyerConePresent:=FALSE;
		sSealConvStatus:=' ';
		bQRSealingConveyorMotor:=FALSE;

		step:=step+1;
		END_IF

	6:	TON_1(IN:=FALSE);
		bSealConvIntOver:=TRUE;
		step:=0;

END_CASE



IF  bIColumnconeDetection  THEN
bConePresent:=TRUE;
ELSE
bConePresent:=FALSE;
END_IF


IF TON_1.ET >t#1ms AND  TON_1.ET<=t#10s THEN
TON_1Running:=TRUE;
ELSE
TON_1Running:=FALSE;
END_IF



TON_1(IN:=bQRSealingConveyorMotor , PT:=T#18s , Q=> , ET=> );

IF bSealConveyerConePresent THEN

HmiConeAtSealConveyer:='Clear Cone At Sealing  Conveyor';
ELSE
HmiConeAtSealConveyer:='   ';
END_IF

(*

IF NOT bIEmergencySwitch or


*)
END_PROGRAM

(* POU StartUp/MatrixConvRst, ST *)
PROGRAM MatrixConvRst
VAR
	step: INT;
	TON_1: TON;
	bConePresent: BOOL;
	TON_1Running: BOOL;
END_VAR
CASE step OF

	0:	 IF bWrpConvIntOver AND bSealConvIntOver  AND bAutoModeOn THEN
		TON_1(IN:=FALSE);
		bQAMatrixConveyor1:=FALSE;
		bQAMatrixConveyor2:=FALSE;
		bQMMatrixConveyorMotor:=FALSE;
		step:=step+1;
		END_IF

	1:  	IF bIRowStopperHome THEN step:=step+1;
		ELSIF NOT bIRowStopperHome THEN bIntRowStopper:=TRUE; step:=step+1; END_IF


	2:	IF bIRowStopperHome THEN  bQRMatrixConveyorMotor:=TRUE;
		bWrpConvIntOver:=FALSE;
		bSealConvIntOver:=FALSE;
		step:=step+1;
		END_IF


	3:	IF bIRowConeDetection THEN
		step:=step+3;
		ELSIF NOT bIRowConeDetection THEN
		step:=step+1;
		END_IF


	4:	IF  TON_1Running  AND bConePresent THEN
		step:=step+1;
		ELSIF TON_1.Q  AND NOT bConePresent THEN
		step:=step+3;
		END_IF



	5:	step:=step+1;


	6:	bQRMatrixConveyorMotor:=FALSE;
		sMatrixConvStatus:='Clear Cone At Matrix Conveyor';
		bConeAtMatrixConveter:=TRUE;
		bConePresent:=FALSE;
		step:=step+2;

	7:	IF NOT bConePresent AND bAutoModeOn   THEN
		bQRMatrixConveyorMotor:=FALSE;
		bConeAtMatrixConveter:=FALSE;

	(*	bRowStopperMoveAftrInt:=TRUE;  *)
		step:=step+1;
		END_IF

	8:	IF  bAutoModeOn(*  bIRowStopper2*)AND bErrorReset   AND NOT bIRowConeDetection  AND bConeAtMatrixConveter  THEN    TON_1(IN:=FALSE); sMatrixConvStatus:='Continue Machine Operation ';
		bMatrixConvIntOver:=TRUE;bConeAtMatrixConveter:=FALSE;
		step:=0;
		ELSIF bAutoModeOn AND  NOT bConeAtMatrixConveter THEN TON_1(IN:=FALSE); sMatrixConvStatus:='Continue Machine Operation ';
		bMatrixConvIntOver:=TRUE;
		step:=0;
		END_IF

END_CASE






IF bIRowConeDetection THEN
bConePresent:=TRUE;
ELSE
bConePresent:=FALSE;
END_IF



IF TON_1.ET >t#1ms AND  TON_1.ET<=t#5s THEN
TON_1Running:=TRUE;
ELSE
TON_1Running:=FALSE;
END_IF

IF bConeAtMatrixConveter THEN

HmiConeAtMatrixConveyer:='Clear Cone At Matrix  Conveyor';
ELSE
HmiConeAtMatrixConveyer:=' Continue Machine Operation';
END_IF


TON_1(IN:=bQRMatrixConveyorMotor , PT:=T#10s , Q=> , ET=> );


IF NOT bIEmergencySwitch OR bStopHmi OR bIMcStop OR bServoOff  THEN
		TON_1(IN:=FALSE);
		bQAMatrixConveyor1:=FALSE;
		bQAMatrixConveyor2:=FALSE;
		bQMMatrixConveyorMotor:=FALSE;
		bIntRowStopper:=FALSE;
		bQRMatrixConveyorMotor:=FALSE;
		TON_1(IN:=FALSE);
		TON_1Running:=FALSE;
		bConePresent:=FALSE;
		bConeAtMatrixConveter:=FALSE;
		bMatrixConvIntOver:=FALSE;
		bMatrixConvIntOver:=FALSE;
		step:=0;
		bConeMiss2AtWrapConv:=FALSE;
END_IF
END_PROGRAM

(* POU SealingUnitRst, ST *)
PROGRAM SealingUnitRst
VAR
	bARWrappingCone123FwdCom: BOOL;
	TON_1: TON;
	step: INT;
	bAR3ConeWrappOver: BOOL;
	tA3ConesealStartDly: TON;
	tA3ConeSealCompDly: TON;
	test: BOOL;
	bFwdRevPistonRst: BOOL;
END_VAR
bQRWrappingChannelPistonValve1:=bARWrappingCone123OnRst;

bQRWrappingChannelPistonValve2:=bARWrappingCone123OnRst;
bQRWrappingChannelPistonValve3:=bARWrappingCone123OnRst;


CASE step OF

	0:	IF  bAutoModeOn AND bAInitializeSeq THEN
		Step:=step+1;
		END_IF


	1:	bQMWrappingChannelPistonValve1:=FALSE;
		bQMWrappingChannelPistonValve2:=FALSE;
		bQMWrappingChannelPistonValve3:=FALSE;
		bQMForwardPistonValve:=FALSE;
		bQMReversePistonValve:=FALSE;
		bAWrappingCone123OnAuto:=FALSE;
		bAWrappingCone123_23OnAuto:=FALSE;
		bAWrappingCone3OnAuto:=FALSE;
		bAWrappingCone23OnAuto:=FALSE;
		bAWrappingCone23OnAuto1:=FALSE;
		bQAForwardPistonValve:=FALSE;
		bQAReversePistonValve:=FALSE;
		bAInitializeSeq:=FALSE;
		Step:=step+1;


	2:	IF NOT bQASealingConveyorMotor THEN
		bFwdRevPistonRst:=TRUE;
		bARWrappingCone123OnRst:=TRUE;
		step:=step+1;
		END_IF


	3:	IF bARWrappingCone123OnRst AND bIWrappingChannelPiston1_End AND bIWrappingChannelPiston2_End AND bIWrappingChannelPiston3_End THEN

		bARWrappingCone123FwdCom:=TRUE;
		TON_1(IN:= FALSE);
		step:=step+1;
		END_IF

	4:	 IF bARWrappingCone123FwdCom THEN
		bARWrappingCone123OnRst:=FALSE;
		step:=step+1;
		END_IF

	5:	bAR3ConeWrappOver:=TRUE;
		step:=step+1;


	6:	IF bAutoModeOn AND  bAR3ConeWrappOver  THEN
		tA3ConesealStartDly(IN:=TRUE , PT:=t#2s , Q=> , ET=> );
		IF tA3ConesealStartDly.Q AND  bIWrappingChannelPiston1_Home  AND bIWrappingChannelPiston2_Home AND bIWrappingChannelPiston3_Home
		 THEN  step:=step+1; END_IF
		END_IF

	7:	IF bAutoModeOn AND   bISealingBottomPistonHome  AND bISealingTopPistonHome AND bISealingSeparatorXAxisHome AND bISealingSeparatorYAxisHome THEN
		bQRSealingSeparatorYAxisPistonValve:=TRUE;
		tA3ConeSealCompDly(IN:=FALSE);

		  step:=step+1;
		END_IF

	8:	IF bAutoModeOn AND  bISealingSeparatorYAxisEnd THEN
		tA3ConesealStartDly(IN:=FALSE);
		bQRSealingTopPistonValve:=TRUE;

		step:=step+1;
		END_IF

	9:	IF bAutoModeOn AND  bISealingTopPistonEnd AND bISealingBottomPistonEnd  THEN
		tA3ConeSealCompDly(IN:=TRUE, PT:= t#2s, Q=> , ET=> );
		IF tA3ConeSealCompDly.Q THEN   step:=step+1; END_IF
		END_IF


	10:	IF bAutoModeOn AND  bISealingTopPistonEnd AND bISealingBottomPistonEnd AND bISealingSeparatorYAxisEnd THEN
		bQRSealingSeparatorXAxisPistonValve:=TRUE;
		step:=step+1;
		END_IF



	11:	IF bAutoModeOn AND  bISealingSeparatorXAxisEnd  THEN
		step:=step+1;
		 END_IF

	12:	bQRSealingTopPistonValve:=FALSE;
		bA3ConeWrappOver:=FALSE;
		bA3ConeWrappOver_24:=FALSE;
		bQRSealingSeparatorYAxisPistonValve:=FALSE;
		bQRSealingSeparatorXAxisPistonValve:=FALSE;
		step:=step+1;

	13:	IF bAutoModeOn AND  bISealingSeparatorXAxisHome AND  bISealingTopPistonHome AND bISealingBottomPistonHome AND bISealingSeparatorYAxisHome  THEN
		bSaelUnitIntOver:=TRUE;
		step:=step+1;
		END_IF

	14:	bSealingUnitIntOver:=TRUE;
		step:=step+1;



	15:	step:=0;



END_CASE

IF bFwdRevPistonRst THEN bQRForwardPistonValve:=TRUE; bQRReversePistonValve:=TRUE; END_IF

IF bIForwardPistonEnd AND bIReversePistonEnd THEN bFwdRevPistonRst:=FALSE; bQRForwardPistonValve:=FALSE; bQRReversePistonValve:=FALSE; END_IF

IF NOT bIEmergencySwitch OR bStopHmi  OR bServoOff  OR bIMcStop THEN

		bQMWrappingChannelPistonValve1:=FALSE;
		bQMWrappingChannelPistonValve2:=FALSE;
		bQMWrappingChannelPistonValve3:=FALSE;
		bQMForwardPistonValve:=FALSE;
		bQMReversePistonValve:=FALSE;
		bAWrappingCone123OnAuto:=FALSE;
		bAWrappingCone123_23OnAuto:=FALSE;
		bAWrappingCone3OnAuto:=FALSE;
		bAWrappingCone23OnAuto:=FALSE;
		bAWrappingCone23OnAuto1:=FALSE;
		bQAForwardPistonValve:=FALSE;
		bQAReversePistonValve:=FALSE;
		bAInitializeSeq:=FALSE;
		bFwdRevPistonRst:=FALSE;
		bARWrappingCone123OnRst:=FALSE;
		bARWrappingCone123FwdCom:=FALSE;
		bAR3ConeWrappOver:=FALSE;
		tA3ConesealStartDly(IN:=FALSE);
		bQRSealingSeparatorXAxisPistonValve:=FALSE;
		bQRSealingSeparatorYAxisPistonValve:=FALSE;
		bQRSealingTopPistonValve:=FALSE;
		bQRSealingTopPistonValve:=FALSE;
		bSaelUnitIntOver:=FALSE;
		step:=0;

END_IF
END_PROGRAM

(* POU Auto/Sealing_Conveyor_23, ST *)
PROGRAM Sealing_Conveyor_23
VAR

	bA3ConeSealStarted23: BOOL;
	bQASealingConveyor1_23: BOOL;
	bQASealingConveyor2_23: BOOL;
	ConvStopDly1_23: TON;
	bA3ConeSealComp23: BOOL;
	step1: INT;
	CTU_1_23: CTU;
	bAConeCountSenEnable1_23: BOOL;
	bA6thConeSealStarted23: BOOL;
	bA6thConeSealComp23: BOOL;
	ConvStopDly2_23: TON;
	step2: INT;
	step3: INT;
	bSealConvIntOverTemp: BOOL;
	bStopHmitemp: BOOL;
	ConeMissChk_1: RS_Error;
	ConeMissErr_1: BOOL;
	ConeMissChk_2: RS_Error;
	ConeMissErr_2: BOOL;
	ConeMissbit: BOOL;
	SealingStep: INT;
	Timer1: TON;
	Timer2: TON;
	Timer3: TON;
	Timer4: TON;
	bAPauseEnable: BOOL;

	bConeMissBit1: BOOL;
	bConeMissBit2: BOOL;
	bConeMissBit3: BOOL;
	bQASealingConveyor3_23: BOOL;
	tSealStopDly: TIME;
	SealingStep2: INT;
	Timer5: TON;
	Timer6: TON;
	Timer7: TON;
	bConeMissBit11: BOOL;
	bConeMissBit22: BOOL;
	bConeMissBit33: BOOL;
	bConeMissBitSec: BOOL;
	tSealStopDlySec: TIME;
	ConeMissMonitorbit: BOOL;
	bAConeMissAtSealConv: BOOL;
	bAConeMissAtSealConv2: BOOL;
	SingleStep: INT;
	TON_6: TON;
	bAConeCountSenSensed: BOOL;
	bAConeCountSenSensedOff: BOOL;
	R_TRIG_3: R_TRIG;
	R_TRIG_9: R_TRIG;
	CTU_AlarmOnly: CTU;
	bCountLock1: BOOL;
	bCountLock2: BOOL;
	bCountLock: BOOL;
	bAConeMissAtSealConv3: BOOL;
	bQASealingConveyor4_23: BOOL;
	bQASealingConveyor5_23: BOOL;
	bAConeMissAtSealConv4: BOOL;
	bQASealingConveyor6_23: BOOL;
	bCountLock3: BOOL;
	bCountLock4: BOOL;
	bCountLock5: BOOL;
	bCountLock6: BOOL;
	bCountLockBit: BOOL;
	bSet1Started: BOOL;
	bSecSetStarted: BOOL;
	SealCountBit2: BOOL;
END_VAR
bQASealingConveyorMotor2:= ((bQASealingConveyor1_23 OR bQASealingConveyor2_23 OR  bQASealingConveyor3_23 OR bQASealingConveyor5_23 OR bQASealingConveyor4_23 OR bQASealingConveyor6_23 )) ;


CASE step1 OF

	0:	IF bAutoModeOn AND b2_3SetHmiSelected AND   bA3ConeWrappOver AND bQASealingSeparatorYAxisPistonValve THEN
		CTU_1_23.RESET:=TRUE;
		CTU_AlarmOnly.RESET:=TRUE;
		bA3ConeSealStarted23:=TRUE;
		ConvStopDly1_23(IN:=FALSE);
		tSealStopDly:=t#1.5s;                                       (* Speed up*)
		step1:=step1+1;
		END_IF

	1:	IF NOT bAPauseSeq THEN step1:=step1+1; END_IF


	2:	IF bAutoModeOn AND b2_3SetHmiSelected AND  bA3ConeSealStarted23 AND bISealingSeparatorXAxisEnd THEN
		bA3ConeSealComp23:=TRUE;
		CTU_1_23.RESET:=FALSE;
		CTU_AlarmOnly.RESET:=FALSE;
		 Timer1(IN:=FALSE);
		step1:=step1+1;
		END_IF

	3:	step1:=step1+1;

	4:	IF bAutoModeOn AND   bA3ConeSealComp23  AND (bSealConvStart1 OR bSealConvStart3 ) AND  NOT bAPauseSeq  AND NOT bASealSepaX_axisRsError THEN
		bQASealingConveyor1_23:=TRUE;
		bSet1Started:=TRUE;
		step1:=step1+1;
		END_IF

	5:	ConvStopDly1_23(IN:=FALSE); step1:=step1+1;


	6:	IF CTU_AlarmOnly.CV>=3 THEN
		bSealConvStart1:=FALSE;
		bSealConvStart3:=FALSE;
		bA3ConeSealComp23:=FALSE;
		bA3ConeSealStarted23:=FALSE;
		bA3COneCrossed:=TRUE;
		step1:=step1+1;
		END_IF

	7:	step1:=step1+1;

	8:	IF bIColumnconeDetection THEN
		step1:=step1+1;
		END_IF

	9:	step1:=step1+1;


	10:	ConvStopDly1_23(IN:=TRUE , PT:= tSealStopDly , Q=> , ET=> );
		IF ConvStopDly1_23.Q THEN    step1:=step1+1; END_IF


	11:	 step1:=step1+1;

	12:	bQASealingConveyor1_23:=FALSE;
		bA3COneCrossed:=FALSE;
		bQASealingConveyor3_23:=FALSE;
		bQASealingConveyor5_23:=FALSE;
		bQASealingConveyor6_23:=FALSE;
		bAColumnPushPistonStart1_23:=TRUE;
		bASealConvEnd1:=TRUE;
		bCountLock1:=FALSE;
		bCountLock5:=FALSE;
		bCountLock6:=FALSE;
		bSet1Started:=FALSE;
		bCountLockBit:=FALSE;
		step1:=step1+1;

	13:	 step1:=step1+1;


	14:	step1:=0;

END_CASE

IF bQASealingConveyorMotor AND bSet1Started  AND CTU_AlarmOnly.CV=3 THEN bCountLockBit:=TRUE; END_IF


IF bQASealingConveyorMotor AND bIConeCountSensor AND b2_3SetHmiSelected AND NOT bCountLockBit AND NOT SealCountBit2  THEN
bAConeCountSenEnable1_23:=TRUE;
ELSE
bAConeCountSenEnable1_23:=FALSE;
END_IF

CTU_1_23(
	CU:=bAConeCountSenEnable1_23 ,
	RESET:= ,
	PV:=6 ,
	Q=> ,
	CV=> );

CTU_AlarmOnly(
	CU:=(bAConeCountSenEnable1_23 AND NOT bCountLock) ,
	RESET:= ,
	PV:=6 ,
	Q=> ,
	CV=> );




CASE step2 OF

	0:	IF bAutoModeOn AND b2_3SetHmiSelected AND  bA6ConeWrappOver23 AND bQASealingSeparatorYAxisPistonValve  THEN
		bA6thConeSealStarted23:=TRUE;
		ConvStopDly2_23(IN:=FALSE);
		tSealStopDlySec:=t#1.5s;                         (* speed up*)
		step2:=step2+1;
		END_IF

	1:	step2:=step2+1;


	2:	 IF   bISealingSeparatorXAxisEnd THEN
		step2:=step2+1;
		END_IF

	3:	 step2:=step2+1;


	4:	IF bAutoModeOn AND b2_3SetHmiSelected  AND bAFirstSetToMatrix   THEN
		bA6thConeSealComp23:=TRUE;
		Timer2(IN:=FALSE); 															(*===============	bAFirstSetToMatrix:=FALSE; ============= Removed for interlock  Checking========= *)
		step2:=step2+1;
		END_IF


	5:	step2:=step2+1;

	6:	IF bAutoModeOn AND   bA6thConeSealComp23  AND  bSealConvStart2 AND  NOT bAPauseSeq THEN
		bQASealingConveyor2_23:=TRUE;
		bSecSetStarted:=TRUE;
		step2:=step2+1;
		END_IF

	7:	ConvStopDly2_23(IN:=FALSE); step2:=step2+1;

	8:	IF CTU_AlarmOnly.CV>=6 THEN
		bSealConvStart2:=FALSE;
		bA6thConeSealComp23:=FALSE;
		bA6thConeSealStarted23:=FALSE;
		bA6ConeCrossed:=TRUE;
		step2:=step2+1;
		END_IF

	9:	 step2:=step2+1;

	10:	IF bIColumnconeDetection THEN
		step2:=step2+1;
		END_IF

	11:	 step2:=step2+1;

	12:	ConvStopDly2_23(IN:=TRUE , PT:=tSealStopDlySec , Q=> , ET=> );
		IF ConvStopDly2_23.Q THEN   step2:=step2+1; END_IF

	13:	 step2:=step2+1;

	14:	 CTU_AlarmOnly.RESET:=TRUE;
		   step2:=step2+1;

	15:	 step2:=step2+1;

	16:	bQASealingConveyor2_23:=FALSE;
		bQASealingConveyor3_23:=FALSE;
		bQASealingConveyor4_23:=FALSE;
		bA6ConeCrossed:=FALSE;
		bAColumnPushPistonStart2_23:=TRUE;
		bASealConvEnd2:=TRUE;
		bCountLock2:=FALSE;
		bCountLock3:=FALSE;
		bCountLock4:=FALSE;
		SealCountBit2:=FALSE;
		bSecSetStarted:=FALSE;
		  step2:=step2+1;

	17:	 step2:=step2+1;

	18:	CTU_AlarmOnly.RESET:=FALSE;
		step2:=0;


END_CASE


IF bQASealingConveyorMotor AND bSecSetStarted AND  CTU_AlarmOnly.CV=6 THEN SealCountBit2:=TRUE; END_IF


(*================ Sealing Conveyor Start Condition=============*)


IF bRowStopperIntOver THEN
bSealConvIntOverTemp:=TRUE;
END_IF




CASE step3 OF


0:	IF bSealConvIntOverTemp  AND b2_3SetHmiSelected  THEN
	Step3:=Step3+1;
	END_IF

